(* IEC 61131-3 sources: std_i2980_v2.06_cp053/Source/IMM/ieccontrol/simulation (part 8) *)

(* ---- ABSafetySimu.pu ---- *)
IMPORT_OVER_LISTFILE
 cTimeSGAutoClose
, cTimeSGAutoOpen
, cTimeSGAutoLock
, cTimeSGAutoUnlock
, cTimeSGAutoFast
, FBEPForceDI
, FBEPUnForceDI
, ABForceDigital
, KSYS_Status
, TON

END_IMPORT

ALGORITHM_BLOCK ABSafetySimu #DUMMY_EDIT_BLOCK

SYSTEM_VAR
 sv_bInitStart : BOOL;
 sv_bSimulate : BOOL;
 sv_ForceSGMoldClose : BOOL;
 sv_ForceSGNozzleClose : BOOL;
 sv_ForceSGNozzleRearClose : BOOL;
 sv_ForceSGRearClose : BOOL;
 sv_ForceEmergencyStop1 : BOOL;
 sv_ForceEmergencyStop2 : BOOL;
 sv_ForceEmergencyStop3 : BOOL;
 sv_ForceEmergencyStop4 : BOOL;
 sv_ForceOilFilterOK : BOOL;
 sv_ForceLightCurtainClose : BOOL;
 sv_ForceSafetyMat : BOOL;
END_VAR

SYSTEM_OBJECT
 TaskSim : TASK;
 PU_Task_13 : TASK;
END_OBJECT

VAR
 fbEPForceDI : FBEPForceDI;
 fbEPUnForceDI : FBEPUnForceDI;
 mbDIEmergencyStop1Linked : BOOL;
 mbDIEmergencyStop2Linked : BOOL;
 mbDIEmergencyStop3Linked : BOOL;
 mbDIEmergencyStop4Linked : BOOL;
 mbDIOilFilterOkLinked : BOOL;
 mbDISGNozzleLinked : BOOL;
 mbDISGNozzleRearLinked : BOOL;
 mbDISGRearLinked : BOOL;
 mbDISGMoldLinked : BOOL;
 mbDISGMoldOpenLinked : BOOL;
 mpbDISGAutoClosed1 : REFTO BOOL;
 mbDISGAutoClosed1Linked : BOOL;
 mpbDISGAutoClosed2 : REFTO BOOL;
 mbDISGAutoClosed2Linked : BOOL;
 mpbDISGAutoOpen : REFTO BOOL;
 mbDISGAutoOpenLinked : BOOL;
 mpbDISGAutoCloseSlow : REFTO BOOL;
 mbDISGAutoCloseSlowLinked : BOOL;
 mbDISGAutoOpenSlowLinked : BOOL;
 mpbDISGAutoLocked : REFTO BOOL;
 mbDISGAutoLockedLinked : BOOL;
 mpbDISGAutoUnlocked : REFTO BOOL;
 mbDISGAutoUnlockedLinked : BOOL;
 mpbDOSGAutoClose : REFTO BOOL;
 mbDOSGAutoCloseLinked : BOOL;
 mpbDOSGAutoFast : REFTO BOOL;
 mbDOSGAutoFastLinked : BOOL;
 mpbDOSGAutoOpen : REFTO BOOL;
 mbDOSGAutoOpenLinked : BOOL;
 mpbDOSGAutoLock : REFTO BOOL;
 mbDOSGAutoLockLinked : BOOL;
 mpbDOSGAutoUnlock : REFTO BOOL;
 mbDOSGAutoUnlockLinked : BOOL;
 mbDISafetyMat1Linked : BOOL;
 mbDISafetyMat2Linked : BOOL;
 mbDILightCurtainClosedLinked : BOOL;
END_VAR

POSTUPDATE_ALGORITHM pStart ON PU_Task_13 WITH sv_bSimulate,sv_bInitStart

#BEGIN_EDIT_BLOCK
(**************************************** WARNING ********************************************
 *** The KEBA Kemro K2 System including software is not intended for safety control tasks! ***
 ***                       For further information see Comment tab!                        ***
 *********************************************************************************************)

IF sv_bSimulate THEN
   START_PROCESS_ALGORITHM(paSimulate);
END_IF;

IF sv_bSimulate AND mbDISGAutoClosed1Linked THEN
   START_PROCESS_ALGORITHM(paSimulateSGAuto);
END_IF;

;#END_EDIT_BLOCK END_ALGORITHM

PROCESS_ALGORITHM paSimulate ON TaskSim

VAR
 fbEPUnForceDI : FBEPUnForceDI;
 mFirstTimeRun : BOOL := TRUE;
 abForceMoldOpenMaxLimitSwitch : ABForceDigital;
 abForceMoldCloseMinLimitSwitch : ABForceDigital;
END_VAR

(* IecGraph-Code *)

(* init step *)
INITIAL_STEP INIT:
aInit (P);
END_STEP

(* steps *)
STEP SIM:
aSimulate (N);
END_STEP

STEP STOP:
aStopSimu (P);
END_STEP

(* transitions *)
TRANSITION SimRequired (* Trans11 *) FROM INIT TO SIM :=  #BEGIN_EDIT_BLOCK
sv_bSimulate
;#END_EDIT_BLOCK
END_TRANSITION

TRANSITION StpSimRequired (* Trans13 *) FROM SIM TO STOP :=  #BEGIN_EDIT_BLOCK
NOT sv_bSimulate
;#END_EDIT_BLOCK
END_TRANSITION

TRANSITION Return (* Trans16 *) FROM STOP TO SIM :=  #BEGIN_EDIT_BLOCK
TRUE
;#END_EDIT_BLOCK
END_TRANSITION

(* end IecGraph-Code *)
(* sfc-code *)

(* stand alone actions *)
ACTION aSimulate: #BEGIN_EDIT_BLOCK
(**************************************** WARNING ********************************************
 *** The KEBA Kemro K2 System including software is not intended for safety control tasks! ***
 ***                       For further information see Comment tab!                        ***
 *********************************************************************************************)

IF mFirstTimeRun THEN
   sv_ForceSGMoldClose := TRUE;
   sv_ForceSGNozzleClose := TRUE;
   sv_ForceSGNozzleRearClose := TRUE;
   sv_ForceSGRearClose := TRUE;
   sv_ForceEmergencyStop1 := TRUE;
   sv_ForceEmergencyStop2 := TRUE;
   sv_ForceEmergencyStop3 := TRUE;
   sv_ForceEmergencyStop4 := TRUE;
   sv_ForceOilFilterOK := FALSE;
   sv_ForceLightCurtainClose := TRUE;
   sv_ForceSafetyMat := TRUE;
   abForceMoldOpenMaxLimitSwitch.aSetForceValue(TRUE);
   abForceMoldCloseMinLimitSwitch.aSetForceValue(TRUE);
   mFirstTimeRun := FALSE;
END_IF;

;#END_EDIT_BLOCK END_ACTION (*aSimulate*)
ACTION aStopSimu: #BEGIN_EDIT_BLOCK
IF mbDIEmergencyStop1Linked THEN
   fbEPUnForceDI(sSysVar := 'OperationMode1.di_EmergencyStop1');
END_IF;
IF mbDIEmergencyStop2Linked THEN
   fbEPUnForceDI(sSysVar := 'OperationMode1.di_EmergencyStop2');
END_IF;
IF mbDIEmergencyStop3Linked THEN
   fbEPUnForceDI(sSysVar := 'OperationMode1.di_EmergencyStop3');
END_IF;
IF mbDIEmergencyStop4Linked THEN
   fbEPUnForceDI(sSysVar := 'OperationMode1.di_EmergencyStop4');
END_IF;

IF mbDIOilFilterOkLinked THEN
   fbEPUnForceDI(sSysVar := 'OilMaintenance1.di_OilFilterOK');
END_IF;

// SG nozzle
IF mbDISGNozzleLinked THEN
   fbEPUnForceDI(sSysVar := 'SafetyGateNozzle1.di_Closed');
END_IF;

// SG nozzle rear
IF mbDISGNozzleRearLinked THEN
   fbEPUnForceDI(sSysVar := 'SafetyGateNozzleRear1.di_Closed');
END_IF;

// SG rear
IF mbDISGRearLinked THEN
   fbEPUnForceDI(sSysVar := 'SafetyGateRear1.di_Closed');
END_IF;

// SG mold
IF mbDISGMoldLinked THEN
   fbEPUnForceDI(sSysVar := 'SafetyGateMold1.di_Closed');
END_IF;
IF mbDISGMoldOpenLinked THEN
   fbEPUnForceDI(sSysVar := 'SafetyGateMold1.di_Open');
END_IF;

IF mbDISafetyMat1Linked THEN
   fbEPUnForceDI(sSysVar := 'SafetyMat1.di_SafetyMat');
END_IF;
IF mbDISafetyMat2Linked THEN
   fbEPUnForceDI(sSysVar := 'SafetyMat2.di_SafetyMat');
END_IF;

IF mbDILightCurtainClosedLinked THEN
   fbEPUnForceDI(sSysVar := 'LightCurtain1.di_Closed');
END_IF;

abForceMoldOpenMaxLimitSwitch.aUnforce();
abForceMoldCloseMinLimitSwitch.aUnforce();

mFirstTimeRun := TRUE;
STOP_PROCESS_ALGORITHM();

;#END_EDIT_BLOCK END_ACTION (*aStopSimu*)
ACTION aInit: #BEGIN_EDIT_BLOCK
(**************************************** WARNING ********************************************
 *** The KEBA Kemro K2 System including software is not intended for safety control tasks! ***
 ***                       For further information see Comment tab!                        ***
 *********************************************************************************************)

abForceMoldOpenMaxLimitSwitch.aInit('Mold1.di_MoldOpenProtect');
abForceMoldCloseMinLimitSwitch.aInit('Mold1.di_MoldCloseProtect');

;#END_EDIT_BLOCK END_ACTION (*aInit*)
(* end sfc-code *)

END_ALGORITHM

POSTUPDATE_ALGORITHM pEmergencyStop ON TaskSim WITH sv_ForceEmergencyStop1,sv_ForceEmergencyStop2,sv_ForceEmergencyStop3,sv_ForceEmergencyStop4,sv_bSimulate

#BEGIN_EDIT_BLOCK
IF sv_bSimulate THEN
   IF mbDIEmergencyStop1Linked THEN
      fbEPForceDI(sSysVar := 'OperationMode1.di_EmergencyStop1', Value := sv_ForceEmergencyStop1);
   END_IF;
   IF mbDIEmergencyStop2Linked THEN
      fbEPForceDI(sSysVar := 'OperationMode1.di_EmergencyStop2', Value := sv_ForceEmergencyStop2);
   END_IF;
   IF mbDIEmergencyStop3Linked THEN
      fbEPForceDI(sSysVar := 'OperationMode1.di_EmergencyStop3', Value := sv_ForceEmergencyStop3);
   END_IF;
   IF mbDIEmergencyStop4Linked THEN
      fbEPForceDI(sSysVar := 'OperationMode1.di_EmergencyStop4', Value := sv_ForceEmergencyStop4);
   END_IF;
END_IF;

;#END_EDIT_BLOCK END_ALGORITHM

POSTUPDATE_ALGORITHM pOilFilterOK ON TaskSim WITH sv_ForceOilFilterOK,sv_bSimulate

#BEGIN_EDIT_BLOCK
IF mbDIOilFilterOkLinked THEN
   IF sv_bSimulate THEN
      fbEPForceDI(sSysVar := 'OilMaintenance1.di_OilFilterOK', Value := sv_ForceOilFilterOK);
   END_IF;
END_IF;

;#END_EDIT_BLOCK END_ALGORITHM

POSTUPDATE_ALGORITHM pSGMoldClose ON TaskSim WITH sv_ForceSGMoldClose,sv_bSimulate

#BEGIN_EDIT_BLOCK
IF sv_bSimulate THEN
   IF mbDISGMoldLinked THEN
      fbEPForceDI(sSysVar :='SafetyGateMold1.di_Closed', Value := sv_ForceSGMoldClose);
   END_IF;
   IF mbDISGMoldOpenLinked THEN
      fbEPForceDI(sSysVar := 'SafetyGateMold1.di_Open', Value := NOT sv_ForceSGMoldClose);
   END_IF;
END_IF;

;#END_EDIT_BLOCK END_ALGORITHM

POSTUPDATE_ALGORITHM pSGNozzleClose ON TaskSim WITH sv_ForceSGNozzleClose,sv_bSimulate

#BEGIN_EDIT_BLOCK
IF sv_bSimulate THEN
   IF mbDISGNozzleLinked THEN
      fbEPForceDI(sSysVar :='SafetyGateNozzle1.di_Closed', Value := sv_ForceSGNozzleClose);
   END_IF;
END_IF;

;#END_EDIT_BLOCK END_ALGORITHM

POSTUPDATE_ALGORITHM pSGNozzleRearClose ON TaskSim WITH sv_ForceSGNozzleRearClose,sv_bSimulate

#BEGIN_EDIT_BLOCK
IF sv_bSimulate THEN
   IF mbDISGNozzleRearLinked THEN
      fbEPForceDI(sSysVar :='SafetyGateNozzleRear1.di_Closed', Value := sv_ForceSGNozzleRearClose);
   END_IF;
END_IF;

;#END_EDIT_BLOCK END_ALGORITHM

POSTUPDATE_ALGORITHM pSGRearClose ON TaskSim WITH sv_ForceSGRearClose,sv_bSimulate

#BEGIN_EDIT_BLOCK
IF sv_bSimulate THEN
   IF mbDISGRearLinked THEN
      fbEPForceDI(sSysVar :='SafetyGateRear1.di_Closed', Value := sv_ForceSGRearClose);
   END_IF;
END_IF;

;#END_EDIT_BLOCK END_ALGORITHM

POSTUPDATE_ALGORITHM pLightCurtainClose ON TaskSim WITH sv_ForceLightCurtainClose,sv_bSimulate

#BEGIN_EDIT_BLOCK
IF sv_bSimulate THEN
   IF mbDILightCurtainClosedLinked THEN
      fbEPForceDI(sSysVar :='LightCurtain1.di_Closed', Value := sv_ForceLightCurtainClose);
   END_IF;
END_IF;

;#END_EDIT_BLOCK END_ALGORITHM

POSTUPDATE_ALGORITHM pSafetyMat ON TaskSim WITH sv_ForceSafetyMat,sv_bSimulate

#BEGIN_EDIT_BLOCK
IF sv_bSimulate THEN
   IF mbDISafetyMat1Linked THEN
      fbEPForceDI(sSysVar :='SafetyMat1.di_SafetyMat', Value := sv_ForceSafetyMat);
   END_IF;
   IF mbDISafetyMat2Linked THEN
      fbEPForceDI(sSysVar :='SafetyMat2.di_SafetyMat', Value := sv_ForceSafetyMat);
   END_IF;
END_IF;

;#END_EDIT_BLOCK END_ALGORITHM

PROCESS_ALGORITHM paInit ON TaskSim AUTOSTART

VAR
 Status : KSYS_Status;
 pbDummy : REFTO BOOL;
END_VAR
#BEGIN_EDIT_BLOCK
pbDummy := GET_SYNC_REFTO('OperationMode1.di_EmergencyStop1', T#0s, Status);
mbDIEmergencyStop1Linked := (Status = KSYS_Status_OK);
pbDummy := GET_SYNC_REFTO('OperationMode1.di_EmergencyStop2', T#0s, Status);
mbDIEmergencyStop2Linked := (Status = KSYS_Status_OK);
pbDummy := GET_SYNC_REFTO('OperationMode1.di_EmergencyStop3', T#0s, Status);
mbDIEmergencyStop3Linked := (Status = KSYS_Status_OK);
pbDummy := GET_SYNC_REFTO('OperationMode1.di_EmergencyStop4', T#0s, Status);
mbDIEmergencyStop4Linked := (Status = KSYS_Status_OK);

pbDummy := GET_SYNC_REFTO('OilMaintenance1.di_OilFilterOK', T#0s, Status);
mbDIOilFilterOkLinked := (Status = KSYS_Status_OK);

pbDummy := GET_SYNC_REFTO('SafetyGateNozzle1.di_Closed', T#0s, Status);
mbDISGNozzleLinked := (Status = KSYS_Status_OK);

(*Optional Safety Gate Nozzle Rear*)
pbDummy := GET_SYNC_REFTO('SafetyGateNozzleRear1.di_Closed', T#0s, Status);
mbDISGNozzleRearLinked := (Status = KSYS_Status_OK);

// Safety Gate Rear
pbDummy := GET_SYNC_REFTO('SafetyGateRear1.di_Closed', T#0s, Status);
mbDISGRearLinked := (Status = KSYS_Status_OK);

// Safety Gate Mold
pbDummy := GET_SYNC_REFTO('SafetyGateMold1.di_Closed', T#0s, Status);
mbDISGMoldLinked := (Status = KSYS_Status_OK);
pbDummy := GET_SYNC_REFTO('SafetyGateMold1.di_Open', T#0s, Status);
mbDISGMoldOpenLinked := (Status = KSYS_Status_OK);

// SafetyGateAuto
mpbDISGAutoClosed1 := GET_SYNC_REFTO('SafetyGateAuto1.di_Closed', T#0s, Status);
mbDISGAutoClosed1Linked := (Status = KSYS_Status_OK);

mpbDISGAutoClosed2 := GET_SYNC_REFTO('SafetyGateAuto1.di_Closed2', T#0s, Status);
mbDISGAutoClosed2Linked := (Status = KSYS_Status_OK);

mpbDISGAutoOpen := GET_SYNC_REFTO('SafetyGateAuto1.di_Open', T#0s, Status);
mbDISGAutoOpenLinked := (Status = KSYS_Status_OK);

mpbDISGAutoCloseSlow := GET_SYNC_REFTO('SafetyGateAuto1.di_CloseSlow', T#0s, Status);
mbDISGAutoCloseSlowLinked := (Status = KSYS_Status_OK);

pbDummy := GET_SYNC_REFTO('SafetyGateAuto1.di_OpenSlow', T#0s, Status);
mbDISGAutoOpenSlowLinked := (Status = KSYS_Status_OK);

mpbDISGAutoLocked := GET_SYNC_REFTO('SafetyGateAuto1.di_Locked', T#0s, Status);
mbDISGAutoLockedLinked := (Status = KSYS_Status_OK);

mpbDISGAutoUnlocked := GET_SYNC_REFTO('SafetyGateAuto1.di_Unlocked', T#0s, Status);
mbDISGAutoUnlockedLinked := (Status = KSYS_Status_OK);

mpbDOSGAutoClose := GET_SYNC_REFTO('SafetyGateAuto1.do_Close', T#0s, Status);
mbDOSGAutoCloseLinked := (Status = KSYS_Status_OK);

mpbDOSGAutoFast := GET_SYNC_REFTO('SafetyGateAuto1.do_Fast', T#0s, Status);
mbDOSGAutoFastLinked := (Status = KSYS_Status_OK);

mpbDOSGAutoOpen := GET_SYNC_REFTO('SafetyGateAuto1.do_Open', T#0s, Status);
mbDOSGAutoOpenLinked := (Status = KSYS_Status_OK);

mpbDOSGAutoLock := GET_SYNC_REFTO('SafetyGateAuto1.do_Lock', T#0s, Status);
mbDOSGAutoLockLinked := (Status = KSYS_Status_OK);

mpbDOSGAutoUnlock := GET_SYNC_REFTO('SafetyGateAuto1.do_Unlock', T#0s, Status);
mbDOSGAutoUnlockLinked := (Status = KSYS_Status_OK);

// SafetyMat
pbDummy := GET_SYNC_REFTO('SafetyMat1.di_SafetyMat', T#0s, Status);
mbDISafetyMat1Linked := (Status = KSYS_Status_OK);

pbDummy := GET_SYNC_REFTO('SafetyMat2.di_SafetyMat', T#0s, Status);
mbDISafetyMat2Linked := (Status = KSYS_Status_OK);

//LightCurtain
pbDummy:= GET_SYNC_REFTO('LightCurtain1.di_Closed', T#0s, Status);
mbDILightCurtainClosedLinked := (Status = KSYS_Status_OK);

STOP_PROCESS_ALGORITHM();

;#END_EDIT_BLOCK END_ALGORITHM

PROCESS_ALGORITHM paSimulateSGAuto ON TaskSim

VAR
 fbTimerSGAutoClose : TON;
 fbTimerSGAutoOpen : TON;
 fbTimerSGAutoLock : TON;
 fbTimerSGAutoUnlock : TON;
 fbTimerSGAutoFast : TON;
 bInitDone : BOOL;
END_VAR

(* IecGraph-Code *)

(* init step *)
INITIAL_STEP INIT:
END_STEP

(* steps *)
STEP SIM:
aSimulate (N);
END_STEP

STEP STOP:
aStopSimu (P);
END_STEP

(* transitions *)
TRANSITION SimRequired (* Trans11 *) FROM INIT TO SIM :=  #BEGIN_EDIT_BLOCK
sv_bSimulate
;#END_EDIT_BLOCK
END_TRANSITION

TRANSITION StpSimRequired (* Trans13 *) FROM SIM TO STOP :=  #BEGIN_EDIT_BLOCK
NOT sv_bSimulate
;#END_EDIT_BLOCK
END_TRANSITION

TRANSITION Return (* Trans16 *) FROM STOP TO SIM :=  #BEGIN_EDIT_BLOCK
TRUE
;#END_EDIT_BLOCK
END_TRANSITION

(* end IecGraph-Code *)
(* sfc-code *)

(* stand alone actions *)
ACTION aStopSimu: #BEGIN_EDIT_BLOCK
IF mbDISGAutoClosed1Linked THEN
   fbEPUnForceDI(sSysVar := 'SafetyGateAuto1.di_Closed');
END_IF;

IF mbDISGAutoClosed2Linked THEN
   fbEPUnForceDI(sSysVar := 'SafetyGateAuto1.di_Closed2');
END_IF;

IF mbDISGAutoOpenLinked THEN
   fbEPUnForceDI(sSysVar := 'SafetyGateAuto1.di_Open');
END_IF;

IF mbDISGAutoOpenSlowLinked THEN
   fbEPUnForceDI(sSysVar := 'SafetyGateAuto1.di_OpenSlow');
END_IF;

IF mbDISGAutoCloseSlowLinked THEN
   fbEPUnForceDI(sSysVar := 'SafetyGateAuto1.di_CloseSlow');
END_IF;

IF mbDISGAutoLockedLinked THEN
   fbEPUnForceDI(sSysVar := 'SafetyGateAuto1.di_Locked');
END_IF;

IF mbDISGAutoUnlockedLinked THEN
   fbEPUnForceDI(sSysVar := 'SafetyGateAuto1.di_Unlocked');
END_IF;

STOP_PROCESS_ALGORITHM();

;#END_EDIT_BLOCK END_ACTION (*aStopSimu*)
ACTION aSimulate: #BEGIN_EDIT_BLOCK
//-------------------------------------------//
// normal movement simulation                //
//-------------------------------------------//

IF NOT bInitDone THEN
   fbEPForceDI(sSysVar := 'SafetyGateAuto1.di_Emergency',Value := TRUE);
   fbEPForceDI(sSysVar := 'SafetyGateAuto1.di_Emergency2',Value := TRUE);

   IF mbDISGAutoClosed1Linked THEN
      fbEPForceDI(sSysVar :='SafetyGateAuto1.di_Closed', Value := FALSE);
   END_IF;
   IF mbDISGAutoClosed2Linked THEN
      fbEPForceDI(sSysVar :='SafetyGateAuto1.di_Closed2', Value := TRUE);
   END_IF;
   IF mbDISGAutoCloseSlowLinked THEN
      fbEPForceDI(sSysVar :='SafetyGateAuto1.di_CloseSlow', Value := FALSE);
   END_IF;

   IF mbDISGAutoOpenLinked THEN
      fbEPForceDI(sSysVar :='SafetyGateAuto1.di_Open', Value := TRUE);
   END_IF;
   IF mbDISGAutoOpenSlowLinked THEN
      fbEPForceDI(sSysVar :='SafetyGateAuto1.di_OpenSlow', Value := TRUE);
   END_IF;

   IF mbDISGAutoLockedLinked THEN
      fbEPForceDI(sSysVar :='SafetyGateAuto1.di_Locked', Value := TRUE);
   END_IF;
   IF mbDISGAutoUnlockedLinked THEN
      fbEPForceDI(sSysVar :='SafetyGateAuto1.di_Unlocked', Value := FALSE);
   END_IF;

   bInitDone := TRUE;
END_IF;

// Safety Gate Close
IF mbDOSGAutoCloseLinked AND mpbDOSGAutoClose^ THEN

   IF mbDISGAutoOpenLinked AND mpbDISGAutoOpen^ THEN
      fbEPForceDI(sSysVar := 'SafetyGateAuto1.di_Open',Value := FALSE);
      fbEPForceDI(sSysVar := 'SafetyGateAuto1.di_OpenSlow',Value := FALSE);
   END_IF;

   IF mbDOSGAutoFastLinked THEN
       fbTimerSGAutoFast (IN := mpbDOSGAutoFast^,
                      PT := cTimeSGAutoFast);
   END_IF;
   IF fbTimerSGAutoFast.Q THEN
      fbTimerSGAutoFast(IN := FALSE);
      fbEPForceDI(sSysVar := 'SafetyGateAuto1.di_CloseSlow',Value := TRUE);
   END_IF;

   fbTimerSGAutoClose (IN := mpbDOSGAutoClose^,
                       PT := cTimeSGAutoClose);
   IF fbTimerSGAutoClose.Q THEN
      fbTimerSGAutoClose(IN := FALSE);
      fbEPForceDI(sSysVar := 'SafetyGateAuto1.di_Closed',Value := TRUE);
      fbEPForceDI(sSysVar := 'SafetyGateAuto1.di_Closed2',Value := FALSE);
   END_IF;
END_IF;

// Safety Gate Open
IF mbDOSGAutoOpenLinked AND mpbDOSGAutoOpen^ THEN
   IF mbDISGAutoClosed1Linked AND mpbDISGAutoClosed1^ THEN
      fbEPForceDI(sSysVar := 'SafetyGateAuto1.di_Closed',Value := FALSE);
      fbEPForceDI(sSysVar := 'SafetyGateAuto1.di_CloseSlow',Value := FALSE);
   END_IF;

   IF mbDISGAutoClosed2Linked AND NOT mpbDISGAutoClosed2^ THEN
      fbEPForceDI(sSysVar := 'SafetyGateAuto1.di_Closed2',Value := TRUE);
   END_IF;

   IF mbDOSGAutoFastLinked THEN
   fbTimerSGAutoFast (IN := mpbDOSGAutoFast^,
                      PT := cTimeSGAutoFast);
   END_IF;
   IF fbTimerSGAutoFast.Q THEN
      fbTimerSGAutoFast(IN := FALSE);
      fbEPForceDI(sSysVar := 'SafetyGateAuto1.di_OpenSlow',Value := TRUE);
   END_IF;

   fbTimerSGAutoOpen (IN := mpbDOSGAutoOpen^,
                       PT := cTimeSGAutoOpen);
   IF fbTimerSGAutoOpen.Q THEN
      fbTimerSGAutoOpen(IN := FALSE);
      fbEPForceDI(sSysVar := 'SafetyGateAuto1.di_Open',Value := TRUE);
   END_IF;
END_IF;

// Safety Gate Lock
IF mbDOSGAutoLockLinked AND mpbDOSGAutoLock^ THEN
   IF mbDISGAutoUnlockedLinked AND mpbDISGAutoUnlocked^ THEN
      fbEPForceDI(sSysVar := 'SafetyGateAuto1.di_Unlocked',Value := FALSE);
   END_IF;

   fbTimerSGAutoLock (IN := mpbDOSGAutoLock^,
                      PT := cTimeSGAutoLock);
   IF fbTimerSGAutoLock.Q THEN
      fbTimerSGAutoLock(IN := TRUE);
      fbEPForceDI(sSysVar := 'SafetyGateAuto1.di_Locked',Value := TRUE);
   END_IF;
END_IF;

// Safety Gate Unlock
IF mbDOSGAutoUnlockLinked AND mpbDOSGAutoUnlock^ THEN
   IF mbDISGAutoLockedLinked AND mpbDISGAutoLocked^ THEN
      fbEPForceDI(sSysVar := 'SafetyGateAuto1.di_Locked',Value := FALSE);
   END_IF;

   fbTimerSGAutoUnlock (IN := mpbDOSGAutoUnlock^,
                        PT := cTimeSGAutoUnlock);
   IF fbTimerSGAutoUnlock.Q THEN
      fbTimerSGAutoUnlock(IN := TRUE);
      fbEPForceDI(sSysVar := 'SafetyGateAuto1.di_Unlocked',Value := TRUE);
   END_IF;
END_IF;

;#END_EDIT_BLOCK END_ACTION (*aSimulate*)
(* end sfc-code *)

END_ALGORITHM

END_ALGORITHM_BLOCK

#END_OF_IEC_PART

@Puma @IecEditor 6 97 @Pou 25
@@@BEG_Comment@@@

@@@END_Comment@@@

@BEG_Contents

@BEG_Func
@RT(17)FuncTreeContainer
0
@END_Func

@BEG_Const
@RT(18)ConstTreeContainer
5
@Var @RT(16)cTimeSGAutoClose @RT(0) @T @F @DT @RT(4)TIME @RT(0) @T @T @BASIC 0 @F
@F @F
@T
@BEG_Attrib
0 @RT(4)t#3s @RT(0)
@END_Attrib
1 1 @F @F @F @F

@Var @RT(15)cTimeSGAutoOpen @RT(0) @T @F @DT @RT(4)TIME @RT(0) @T @T @BASIC 0 @F
@F @F
@T
@BEG_Attrib
0 @RT(4)t#3s @RT(0)
@END_Attrib
1 1 @F @F @F @F

@Var @RT(15)cTimeSGAutoLock @RT(0) @T @F @DT @RT(4)TIME @RT(0) @T @T @BASIC 0 @F
@F @F
@T
@BEG_Attrib
0 @RT(4)t#1s @RT(0)
@END_Attrib
1 1 @F @F @F @F

@Var @RT(17)cTimeSGAutoUnlock @RT(0) @T @F @DT @RT(4)TIME @RT(0) @T @T @BASIC 0 @F
@F @F
@T
@BEG_Attrib
0 @RT(4)t#1s @RT(0)
@END_Attrib
1 1 @F @F @F @F

@Var @RT(15)cTimeSGAutoFast @RT(0) @T @F @DT @RT(4)TIME @RT(0) @T @T @BASIC 0 @F
@F @F
@T
@BEG_Attrib
0 @RT(4)t#2s @RT(0)
@END_Attrib
1 1 @F @F @F @F

@END_Const

@BEG_Export

@BEG_Kind
@ALGORITHM_BLOCK @RT(12)ABSafetySimu @STRUCTURED_TEXT
@RT(0) @RT(0) @RT(0)
@END_Kind

@BEG_Dcl
@RT(16)DclTreeContainer
53
@Var @RT(7)TaskSim @RT(0) @T @T @RENAMED 0 @T @T @DT @RT(4)TASK @RT(0) @T @T @BASIC 0 @F
@F @F
@T
@BEG_Attrib
3 @RT(0) @RT(0) @RT(0)
@END_Attrib
1 7 @F @F @F @F

@Var @RT(10)PU_Task_13 @RT(0) @T @T @RENAMED 0 @T @T @DT @RT(4)TASK @RT(0) @T @T @BASIC 0 @F
@F @F
@T
@BEG_Attrib
3 @RT(0) @RT(0) @RT(0)
@END_Attrib
1 7 @F @F @F @F

@Var @RT(13)sv_bInitStart @RT(0) @T @F @DT @RT(4)BOOL @RT(0) @T @T @BASIC 0 @F
@F @F
@T
@BEG_Attrib
3 @RT(0) @RT(0) @RT(0)
@END_Attrib
1 8 @F @F @F @F

@Var @RT(12)sv_bSimulate @RT(0) @T @F @DT @RT(4)BOOL @RT(0) @T @T @BASIC 0 @F
@F @F
@T
@BEG_Attrib
3 @RT(0) @RT(0) @RT(0)
@END_Attrib
1 8 @F @F @F @F

@Var @RT(11)fbEPForceDI @RT(0) @T @T @DERIVED 0 @T @T @DT @RT(11)FBEPForceDI @RT(0) @T @T @UNKNOWN 0 @F
@F @F
@T
@BEG_Attrib
3 @RT(0) @RT(0) @RT(0)
@END_Attrib
1 0 @F @F @F @F

@Var @RT(13)fbEPUnForceDI @RT(0) @T @T @DERIVED 0 @T @T @DT @RT(13)FBEPUnForceDI @RT(0) @T @T @UNKNOWN 0 @F
@F @F
@T
@BEG_Attrib
3 @RT(0) @RT(0) @RT(0)
@END_Attrib
1 0 @F @F @F @F

@Var @RT(19)sv_ForceSGMoldClose @RT(0) @T @F @DT @RT(4)BOOL @RT(0) @T @T @BASIC 0 @F
@F @F
@T
@BEG_Attrib
3 @RT(0) @RT(0) @RT(0)
@END_Attrib
1 8 @F @F @F @F

@Var @RT(21)sv_ForceSGNozzleClose @RT(0) @T @F @DT @RT(4)BOOL @RT(0) @T @T @BASIC 0 @F
@F @F
@T
@BEG_Attrib
3 @RT(0) @RT(0) @RT(0)
@END_Attrib
1 8 @F @F @F @F

@Var @RT(25)sv_ForceSGNozzleRearClose @RT(0) @T @F @DT @RT(4)BOOL @RT(0) @T @T @BASIC 0 @F
@F @F
@T
@BEG_Attrib
3 @RT(0) @RT(0) @RT(0)
@END_Attrib
1 8 @F @F @F @F

@Var @RT(19)sv_ForceSGRearClose @RT(0) @T @F @DT @RT(4)BOOL @RT(0) @T @T @BASIC 0 @F
@F @F
@T
@BEG_Attrib
3 @RT(0) @RT(0) @RT(0)
@END_Attrib
1 8 @F @F @F @F

@Var @RT(22)sv_ForceEmergencyStop1 @RT(0) @T @F @DT @RT(4)BOOL @RT(0) @T @T @BASIC 0 @F
@F @F
@T
@BEG_Attrib
3 @RT(0) @RT(0) @RT(0)
@END_Attrib
1 8 @F @F @F @F

@Var @RT(22)sv_ForceEmergencyStop2 @RT(0) @T @F @DT @RT(4)BOOL @RT(0) @T @T @BASIC 0 @F
@F @F
@T
@BEG_Attrib
3 @RT(0) @RT(0) @RT(0)
@END_Attrib
1 8 @F @F @F @F

@Var @RT(22)sv_ForceEmergencyStop3 @RT(0) @T @F @DT @RT(4)BOOL @RT(0) @T @T @BASIC 0 @F
@F @F
@T
@BEG_Attrib
3 @RT(0) @RT(0) @RT(0)
@END_Attrib
1 8 @F @F @F @F

@Var @RT(22)sv_ForceEmergencyStop4 @RT(0) @T @F @DT @RT(4)BOOL @RT(0) @T @T @BASIC 0 @F
@F @F
@T
@BEG_Attrib
3 @RT(0) @RT(0) @RT(0)
@END_Attrib
1 8 @F @F @F @F

@Var @RT(19)sv_ForceOilFilterOK @RT(0) @T @F @DT @RT(4)BOOL @RT(0) @T @T @BASIC 0 @F
@F @F
@T
@BEG_Attrib
3 @RT(0) @RT(0) @RT(0)
@END_Attrib
1 8 @F @F @F @F

@Var @RT(25)sv_ForceLightCurtainClose @RT(0) @T @T @RENAMED 0 @T @T @DT @RT(4)BOOL @RT(0) @T @T @BASIC 0 @F
@F @F
@T
@BEG_Attrib
3 @RT(0) @RT(0) @RT(0)
@END_Attrib
1 8 @F @F @F @F

@Var @RT(17)sv_ForceSafetyMat @RT(0) @T @T @RENAMED 0 @T @T @DT @RT(4)BOOL @RT(0) @T @T @BASIC 0 @F
@F @F
@T
@BEG_Attrib
3 @RT(0) @RT(0) @RT(0)
@END_Attrib
1 8 @F @F @F @F

@Var @RT(24)mbDIEmergencyStop1Linked @RT(0) @T @F @DT @RT(4)BOOL @RT(0) @T @T @BASIC 0 @F
@F @F
@T
@BEG_Attrib
3 @RT(0) @RT(0) @RT(0)
@END_Attrib
1 0 @F @F @F @F

@Var @RT(24)mbDIEmergencyStop2Linked @RT(0) @T @F @DT @RT(4)BOOL @RT(0) @T @T @BASIC 0 @F
@F @F
@T
@BEG_Attrib
3 @RT(0) @RT(0) @RT(0)
@END_Attrib
1 0 @F @F @F @F

@Var @RT(24)mbDIEmergencyStop3Linked @RT(0) @T @F @DT @RT(4)BOOL @RT(0) @T @T @BASIC 0 @F
@F @F
@T
@BEG_Attrib
3 @RT(0) @RT(0) @RT(0)
@END_Attrib
1 0 @F @F @F @F

@Var @RT(24)mbDIEmergencyStop4Linked @RT(0) @T @F @DT @RT(4)BOOL @RT(0) @T @T @BASIC 0 @F
@F @F
@T
@BEG_Attrib
3 @RT(0) @RT(0) @RT(0)
@END_Attrib
1 0 @F @F @F @F

@Var @RT(21)mbDIOilFilterOkLinked @RT(0) @T @F @DT @RT(4)BOOL @RT(0) @T @T @BASIC 0 @F
@F @F
@T
@BEG_Attrib
3 @RT(0) @RT(0) @RT(0)
@END_Attrib
1 0 @F @F @F @F

@Var @RT(18)mbDISGNozzleLinked @RT(0) @T @F @DT @RT(4)BOOL @RT(0) @T @T @BASIC 0 @F
@F @F
@T
@BEG_Attrib
3 @RT(0) @RT(0) @RT(0)
@END_Attrib
1 0 @F @F @F @F

@Var @RT(22)mbDISGNozzleRearLinked @RT(0) @T @F @DT @RT(4)BOOL @RT(0) @T @T @BASIC 0 @F
@F @F
@T
@BEG_Attrib
3 @RT(0) @RT(0) @RT(0)
@END_Attrib
1 0 @F @F @F @F

@Var @RT(16)mbDISGRearLinked @RT(0) @T @F @DT @RT(4)BOOL @RT(0) @T @T @BASIC 0 @F
@F @F
@T
@BEG_Attrib
3 @RT(0) @RT(0) @RT(0)
@END_Attrib
1 0 @F @F @F @F

@Var @RT(16)mbDISGMoldLinked @RT(0) @T @F @DT @RT(4)BOOL @RT(0) @T @T @BASIC 0 @F
@F @F
@T
@BEG_Attrib
3 @RT(0) @RT(0) @RT(0)
@END_Attrib
1 0 @F @F @F @F

@Var @RT(20)mbDISGMoldOpenLinked @RT(0) @T @F @DT @RT(4)BOOL @RT(0) @T @T @BASIC 0 @F
@F @F
@T
@BEG_Attrib
3 @RT(0) @RT(0) @RT(0)
@END_Attrib
1 0 @F @F @F @F

@Var @RT(18)mpbDISGAutoClosed1 @RT(0) @T @T @REFTO 0 @T @DT @RT(4)BOOL @RT(0) @T @T @BASIC 0 @F
@F @F
@T
@BEG_Attrib
3 @RT(0) @RT(0) @RT(0)
@END_Attrib
1 0 @F @F @F @F

@Var @RT(23)mbDISGAutoClosed1Linked @RT(0) @T @F @DT @RT(4)BOOL @RT(0) @T @T @BASIC 0 @F
@F @F
@T
@BEG_Attrib
3 @RT(0) @RT(0) @RT(0)
@END_Attrib
1 0 @F @F @F @F

@Var @RT(18)mpbDISGAutoClosed2 @RT(0) @T @T @REFTO 0 @T @DT @RT(4)BOOL @RT(0) @T @T @BASIC 0 @F
@F @F
@T
@BEG_Attrib
3 @RT(0) @RT(0) @RT(0)
@END_Attrib
1 0 @F @F @F @F

@Var @RT(23)mbDISGAutoClosed2Linked @RT(0) @T @F @DT @RT(4)BOOL @RT(0) @T @T @BASIC 0 @F
@F @F
@T
@BEG_Attrib
3 @RT(0) @RT(0) @RT(0)
@END_Attrib
1 0 @F @F @F @F

@Var @RT(15)mpbDISGAutoOpen @RT(0) @T @T @REFTO 0 @T @DT @RT(4)BOOL @RT(0) @T @T @BASIC 0 @F
@F @F
@T
@BEG_Attrib
3 @RT(0) @RT(0) @RT(0)
@END_Attrib
1 0 @F @F @F @F

@Var @RT(20)mbDISGAutoOpenLinked @RT(0) @T @F @DT @RT(4)BOOL @RT(0) @T @T @BASIC 0 @F
@F @F
@T
@BEG_Attrib
3 @RT(0) @RT(0) @RT(0)
@END_Attrib
1 0 @F @F @F @F

@Var @RT(20)mpbDISGAutoCloseSlow @RT(0) @T @T @REFTO 0 @T @DT @RT(4)BOOL @RT(0) @T @T @BASIC 0 @F
@F @F
@T
@BEG_Attrib
3 @RT(0) @RT(0) @RT(0)
@END_Attrib
1 0 @F @F @F @F

@Var @RT(25)mbDISGAutoCloseSlowLinked @RT(0) @T @F @DT @RT(4)BOOL @RT(0) @T @T @BASIC 0 @F
@F @F
@T
@BEG_Attrib
3 @RT(0) @RT(0) @RT(0)
@END_Attrib
1 0 @F @F @F @F

@Var @RT(24)mbDISGAutoOpenSlowLinked @RT(0) @T @F @DT @RT(4)BOOL @RT(0) @T @T @BASIC 0 @F
@F @F
@T
@BEG_Attrib
3 @RT(0) @RT(0) @RT(0)
@END_Attrib
1 0 @F @F @F @F

@Var @RT(17)mpbDISGAutoLocked @RT(0) @T @T @REFTO 0 @T @DT @RT(4)BOOL @RT(0) @T @T @BASIC 0 @F
@F @F
@T
@BEG_Attrib
3 @RT(0) @RT(0) @RT(0)
@END_Attrib
1 0 @F @F @F @F

@Var @RT(22)mbDISGAutoLockedLinked @RT(0) @T @F @DT @RT(4)BOOL @RT(0) @T @T @BASIC 0 @F
@F @F
@T
@BEG_Attrib
3 @RT(0) @RT(0) @RT(0)
@END_Attrib
1 0 @F @F @F @F

@Var @RT(19)mpbDISGAutoUnlocked @RT(0) @T @T @REFTO 0 @T @DT @RT(4)BOOL @RT(0) @T @T @BASIC 0 @F
@F @F
@T
@BEG_Attrib
3 @RT(0) @RT(0) @RT(0)
@END_Attrib
1 0 @F @F @F @F

@Var @RT(24)mbDISGAutoUnlockedLinked @RT(0) @T @F @DT @RT(4)BOOL @RT(0) @T @T @BASIC 0 @F
@F @F
@T
@BEG_Attrib
3 @RT(0) @RT(0) @RT(0)
@END_Attrib
1 0 @F @F @F @F

@Var @RT(16)mpbDOSGAutoClose @RT(0) @T @T @REFTO 0 @T @DT @RT(4)BOOL @RT(0) @T @T @BASIC 0 @F
@F @F
@T
@BEG_Attrib
3 @RT(0) @RT(0) @RT(0)
@END_Attrib
1 0 @F @F @F @F

@Var @RT(21)mbDOSGAutoCloseLinked @RT(0) @T @F @DT @RT(4)BOOL @RT(0) @T @T @BASIC 0 @F
@F @F
@T
@BEG_Attrib
3 @RT(0) @RT(0) @RT(0)
@END_Attrib
1 0 @F @F @F @F

@Var @RT(15)mpbDOSGAutoFast @RT(0) @T @T @REFTO 0 @T @DT @RT(4)BOOL @RT(0) @T @T @BASIC 0 @F
@F @F
@T
@BEG_Attrib
3 @RT(0) @RT(0) @RT(0)
@END_Attrib
1 0 @F @F @F @F

@Var @RT(20)mbDOSGAutoFastLinked @RT(0) @T @F @DT @RT(4)BOOL @RT(0) @T @T @BASIC 0 @F
@F @F
@T
@BEG_Attrib
3 @RT(0) @RT(0) @RT(0)
@END_Attrib
1 0 @F @F @F @F

@Var @RT(15)mpbDOSGAutoOpen @RT(0) @T @T @REFTO 0 @T @DT @RT(4)BOOL @RT(0) @T @T @BASIC 0 @F
@F @F
@T
@BEG_Attrib
3 @RT(0) @RT(0) @RT(0)
@END_Attrib
1 0 @F @F @F @F

@Var @RT(20)mbDOSGAutoOpenLinked @RT(0) @T @F @DT @RT(4)BOOL @RT(0) @T @T @BASIC 0 @F
@F @F
@T
@BEG_Attrib
3 @RT(0) @RT(0) @RT(0)
@END_Attrib
1 0 @F @F @F @F

@Var @RT(15)mpbDOSGAutoLock @RT(0) @T @T @REFTO 0 @T @DT @RT(4)BOOL @RT(0) @T @T @BASIC 0 @F
@F @F
@T
@BEG_Attrib
3 @RT(0) @RT(0) @RT(0)
@END_Attrib
1 0 @F @F @F @F

@Var @RT(20)mbDOSGAutoLockLinked @RT(0) @T @F @DT @RT(4)BOOL @RT(0) @T @T @BASIC 0 @F
@F @F
@T
@BEG_Attrib
3 @RT(0) @RT(0) @RT(0)
@END_Attrib
1 0 @F @F @F @F

@Var @RT(17)mpbDOSGAutoUnlock @RT(0) @T @T @REFTO 0 @T @DT @RT(4)BOOL @RT(0) @T @T @BASIC 0 @F
@F @F
@T
@BEG_Attrib
3 @RT(0) @RT(0) @RT(0)
@END_Attrib
1 0 @F @F @F @F

@Var @RT(22)mbDOSGAutoUnlockLinked @RT(0) @T @F @DT @RT(4)BOOL @RT(0) @T @T @BASIC 0 @F
@F @F
@T
@BEG_Attrib
3 @RT(0) @RT(0) @RT(0)
@END_Attrib
1 0 @F @F @F @F

@Var @RT(20)mbDISafetyMat1Linked @RT(0) @T @F @DT @RT(4)BOOL @RT(0) @T @T @BASIC 0 @F
@F @F
@T
@BEG_Attrib
3 @RT(0) @RT(0) @RT(0)
@END_Attrib
1 0 @F @F @F @F

@Var @RT(20)mbDISafetyMat2Linked @RT(0) @T @F @DT @RT(4)BOOL @RT(0) @T @T @BASIC 0 @F
@F @F
@T
@BEG_Attrib
3 @RT(0) @RT(0) @RT(0)
@END_Attrib
1 0 @F @F @F @F

@Var @RT(28)mbDILightCurtainClosedLinked @RT(0) @T @F @DT @RT(4)BOOL @RT(0) @T @T @BASIC 0 @F
@F @F
@T
@BEG_Attrib
3 @RT(0) @RT(0) @RT(0)
@END_Attrib
1 0 @F @F @F @F

@END_Dcl

@END_Export

@BEG_Body

12

@BEG_Export

@BEG_Algo
@POSTUPDATE_ALGORITHM @RT(6)pStart @STRUCTURED_TEXT
@RT(0) @RT(26)sv_bSimulate,sv_bInitStart @RT(10)PU_Task_13 @F @F
@END_Algo

@BEG_Dcl
@RT(16)DclTreeContainer
0
@END_Dcl

@END_Export

@BEG_Export

@BEG_Algo
@PROCESS_ALGORITHM @RT(10)paSimulate @SEQUENTIAL_FLOW_CHART
@RT(0) @RT(0) @RT(7)TaskSim @F @F
@END_Algo

@BEG_Dcl
@RT(16)DclTreeContainer
4
@Var @RT(13)fbEPUnForceDI @RT(0) @T @T @DERIVED 0 @T @T @DT @RT(13)FBEPUnForceDI @RT(0) @T @T @UNKNOWN 0 @F
@F @F
@T
@BEG_Attrib
3 @RT(0) @RT(0) @RT(0)
@END_Attrib
1 0 @F @F @F @F

@Var @RT(13)mFirstTimeRun @RT(0) @T @F @DT @RT(4)BOOL @RT(0) @T @T @BASIC 0 @F
@F @F
@T
@BEG_Attrib
3 @RT(4)TRUE @RT(0) @RT(0)
@END_Attrib
1 0 @F @F @F @F

@Var @RT(29)abForceMoldOpenMaxLimitSwitch @RT(0) @T @T @DERIVED 0 @F @RT(14)ABForceDigital @F
@T
@BEG_Attrib
3 @RT(0) @RT(0) @RT(0)
@END_Attrib
1 0 @F @F @F @F

@Var @RT(30)abForceMoldCloseMinLimitSwitch @RT(0) @T @T @DERIVED 0 @F @RT(14)ABForceDigital @F
@T
@BEG_Attrib
3 @RT(0) @RT(0) @RT(0)
@END_Attrib
1 0 @F @F @F @F

@END_Dcl

@END_Export

@BEG_Export

@BEG_Algo
@POSTUPDATE_ALGORITHM @RT(14)pEmergencyStop @STRUCTURED_TEXT
@RT(0) @RT(104)sv_ForceEmergencyStop1,sv_ForceEmergencyStop2,sv_ForceEmergencyStop3,sv_ForceEmergencyStop4,sv_bSimulate @RT(7)TaskSim @F @F
@END_Algo

@BEG_Dcl
@RT(16)DclTreeContainer
0
@END_Dcl

@END_Export

@BEG_Export

@BEG_Algo
@POSTUPDATE_ALGORITHM @RT(12)pOilFilterOK @STRUCTURED_TEXT
@RT(0) @RT(32)sv_ForceOilFilterOK,sv_bSimulate @RT(7)TaskSim @F @F
@END_Algo

@BEG_Dcl
@RT(16)DclTreeContainer
0
@END_Dcl

@END_Export

@BEG_Export

@BEG_Algo
@POSTUPDATE_ALGORITHM @RT(12)pSGMoldClose @STRUCTURED_TEXT
@RT(0) @RT(32)sv_ForceSGMoldClose,sv_bSimulate @RT(7)TaskSim @F @F
@END_Algo

@BEG_Dcl
@RT(16)DclTreeContainer
0
@END_Dcl

@END_Export

@BEG_Export

@BEG_Algo
@POSTUPDATE_ALGORITHM @RT(14)pSGNozzleClose @STRUCTURED_TEXT
@RT(0) @RT(34)sv_ForceSGNozzleClose,sv_bSimulate @RT(7)TaskSim @F @F
@END_Algo

@BEG_Dcl
@RT(16)DclTreeContainer
0
@END_Dcl

@END_Export

@BEG_Export

@BEG_Algo
@POSTUPDATE_ALGORITHM @RT(18)pSGNozzleRearClose @STRUCTURED_TEXT
@RT(0) @RT(38)sv_ForceSGNozzleRearClose,sv_bSimulate @RT(7)TaskSim @F @F
@END_Algo

@BEG_Dcl
@RT(16)DclTreeContainer
0
@END_Dcl

@END_Export

@BEG_Export

@BEG_Algo
@POSTUPDATE_ALGORITHM @RT(12)pSGRearClose @STRUCTURED_TEXT
@RT(0) @RT(32)sv_ForceSGRearClose,sv_bSimulate @RT(7)TaskSim @F @F
@END_Algo

@BEG_Dcl
@RT(16)DclTreeContainer
0
@END_Dcl

@END_Export

@BEG_Export

@BEG_Algo
@POSTUPDATE_ALGORITHM @RT(18)pLightCurtainClose @STRUCTURED_TEXT
@RT(0) @RT(38)sv_ForceLightCurtainClose,sv_bSimulate @RT(7)TaskSim @F @F
@END_Algo

@BEG_Dcl
@RT(16)DclTreeContainer
0
@END_Dcl

@END_Export

@BEG_Export

@BEG_Algo
@POSTUPDATE_ALGORITHM @RT(10)pSafetyMat @STRUCTURED_TEXT
@RT(0) @RT(30)sv_ForceSafetyMat,sv_bSimulate @RT(7)TaskSim @F @F
@END_Algo

@BEG_Dcl
@RT(16)DclTreeContainer
0
@END_Dcl

@END_Export

@BEG_Export

@BEG_Algo
@PROCESS_ALGORITHM @RT(6)paInit @STRUCTURED_TEXT
@RT(0) @RT(0) @RT(7)TaskSim @T @F
@END_Algo

@BEG_Dcl
@RT(16)DclTreeContainer
2
@Var @RT(6)Status @RT(0) @T @T @DERIVED 0 @T @T @DT @RT(11)KSYS_Status @RT(0) @T @T @UNKNOWN 0 @F
@F @F
@T
@BEG_Attrib
3 @RT(0) @RT(0) @RT(0)
@END_Attrib
1 0 @F @F @F @F

@Var @RT(7)pbDummy @RT(0) @T @T @REFTO 0 @T @DT @RT(4)BOOL @RT(0) @T @T @BASIC 0 @F
@F @F
@T
@BEG_Attrib
3 @RT(0) @RT(0) @RT(0)
@END_Attrib
1 0 @F @F @F @F

@END_Dcl

@END_Export

@BEG_Export

@BEG_Algo
@PROCESS_ALGORITHM @RT(16)paSimulateSGAuto @SEQUENTIAL_FLOW_CHART
@RT(0) @RT(0) @RT(7)TaskSim @F @F
@END_Algo

@BEG_Dcl
@RT(16)DclTreeContainer
6
@Var @RT(18)fbTimerSGAutoClose @RT(0) @T @T @DERIVED 0 @T @T @DT @RT(3)TON @RT(0) @T @T @UNKNOWN 0 @F
@F @F
@T
@BEG_Attrib
3 @RT(0) @RT(0) @RT(0)
@END_Attrib
1 0 @F @F @F @F

@Var @RT(17)fbTimerSGAutoOpen @RT(0) @T @T @DERIVED 0 @T @T @DT @RT(3)TON @RT(0) @T @T @UNKNOWN 0 @F
@F @F
@T
@BEG_Attrib
3 @RT(0) @RT(0) @RT(0)
@END_Attrib
1 0 @F @F @F @F

@Var @RT(17)fbTimerSGAutoLock @RT(0) @T @T @DERIVED 0 @T @T @DT @RT(3)TON @RT(0) @T @T @UNKNOWN 0 @F
@F @F
@T
@BEG_Attrib
3 @RT(0) @RT(0) @RT(0)
@END_Attrib
1 0 @F @F @F @F

@Var @RT(19)fbTimerSGAutoUnlock @RT(0) @T @T @DERIVED 0 @T @T @DT @RT(3)TON @RT(0) @T @T @UNKNOWN 0 @F
@F @F
@T
@BEG_Attrib
3 @RT(0) @RT(0) @RT(0)
@END_Attrib
1 0 @F @F @F @F

@Var @RT(17)fbTimerSGAutoFast @RT(0) @T @T @DERIVED 0 @T @T @DT @RT(3)TON @RT(0) @T @T @UNKNOWN 0 @F
@F @F
@T
@BEG_Attrib
3 @RT(0) @RT(0) @RT(0)
@END_Attrib
1 0 @F @F @F @F

@Var @RT(9)bInitDone @RT(0) @T @F @DT @RT(4)BOOL @RT(0) @T @T @BASIC 0 @F
@F @F
@T
@BEG_Attrib
3 @RT(0) @RT(0) @RT(0)
@END_Attrib
1 0 @F @F @F @F

@END_Dcl

@END_Export

@BEG_Body
@TL(13)
(**************************************** WARNING ********************************************
 *** The KEBA Kemro K2 System including software is not intended for safety control tasks! ***
 ***                       For further information see Comment tab!                        ***
 *********************************************************************************************)

IF sv_bSimulate THEN
   START_PROCESS_ALGORITHM(paSimulate);
END_IF;

IF sv_bSimulate AND mbDISGAutoClosed1Linked THEN
   START_PROCESS_ALGORITHM(paSimulateSGAuto);
END_IF;

@END_Body

@@@BEG_Comment@@@
@TL(0)

@@@END_Comment@@@

@BEG_SfcBody
16 13 17

@BEG_SfcData 2
@StepSeq @RT(4)sseq @F 3
@Step @RT(4)INIT @F @T @F @F @RT(0) @F
@AcbCont @RT(7)unnamed @F 1
@Acb @RT(5)aInit @F @F @RT(1)P @RT(0) @F @F @F @F

@Trans @RT(11)SimRequired @F @T @F @F @T @T @TL(2)
sv_bSimulate

@RT(7)Trans11 @F
@Loop @RT(4)loop @F 2
@StepSeq @RT(3)seq @F 3
@Step @RT(3)SIM @F @F @F @F @RT(0) @F
@AcbCont @RT(7)unnamed @F 1
@Acb @RT(9)aSimulate @F @F @RT(1)N @RT(0) @F @F @T @F

@Trans @RT(14)StpSimRequired @F @T @F @F @T @T @TL(2)
NOT sv_bSimulate

@RT(7)Trans13 @F
@Step @RT(4)STOP @F @F @F @F @RT(0) @F
@AcbCont @RT(7)unnamed @F 1
@Acb @RT(9)aStopSimu @F @F @RT(1)P @RT(0) @F @F @T @F

@Trans @RT(6)Return @F @T @T @T @T @T @TL(2)
TRUE

@RT(7)Trans16 @F

@END_SfcData
@SaActions 3
@SaText @RT(9)aSimulate 1 @TL(22)
(**************************************** WARNING ********************************************
 *** The KEBA Kemro K2 System including software is not intended for safety control tasks! ***
 ***                       For further information see Comment tab!                        ***
 *********************************************************************************************)

IF mFirstTimeRun THEN
   sv_ForceSGMoldClose := TRUE;
   sv_ForceSGNozzleClose := TRUE;
   sv_ForceSGNozzleRearClose := TRUE;
   sv_ForceSGRearClose := TRUE;
   sv_ForceEmergencyStop1 := TRUE;
   sv_ForceEmergencyStop2 := TRUE;
   sv_ForceEmergencyStop3 := TRUE;
   sv_ForceEmergencyStop4 := TRUE;
   sv_ForceOilFilterOK := FALSE;
   sv_ForceLightCurtainClose := TRUE;
   sv_ForceSafetyMat := TRUE;
   abForceMoldOpenMaxLimitSwitch.aSetForceValue(TRUE);
   abForceMoldCloseMinLimitSwitch.aSetForceValue(TRUE);
   mFirstTimeRun := FALSE;
END_IF;

@SaText @RT(9)aStopSimu 1 @TL(57)
IF mbDIEmergencyStop1Linked THEN
   fbEPUnForceDI(sSysVar := 'OperationMode1.di_EmergencyStop1');
END_IF;
IF mbDIEmergencyStop2Linked THEN
   fbEPUnForceDI(sSysVar := 'OperationMode1.di_EmergencyStop2');
END_IF;
IF mbDIEmergencyStop3Linked THEN
   fbEPUnForceDI(sSysVar := 'OperationMode1.di_EmergencyStop3');
END_IF;
IF mbDIEmergencyStop4Linked THEN
   fbEPUnForceDI(sSysVar := 'OperationMode1.di_EmergencyStop4');
END_IF;

IF mbDIOilFilterOkLinked THEN
   fbEPUnForceDI(sSysVar := 'OilMaintenance1.di_OilFilterOK');
END_IF;

// SG nozzle
IF mbDISGNozzleLinked THEN
   fbEPUnForceDI(sSysVar := 'SafetyGateNozzle1.di_Closed');
END_IF;

// SG nozzle rear
IF mbDISGNozzleRearLinked THEN
   fbEPUnForceDI(sSysVar := 'SafetyGateNozzleRear1.di_Closed');
END_IF;

// SG rear
IF mbDISGRearLinked THEN
   fbEPUnForceDI(sSysVar := 'SafetyGateRear1.di_Closed');
END_IF;

// SG mold
IF mbDISGMoldLinked THEN
   fbEPUnForceDI(sSysVar := 'SafetyGateMold1.di_Closed');
END_IF;
IF mbDISGMoldOpenLinked THEN
   fbEPUnForceDI(sSysVar := 'SafetyGateMold1.di_Open');
END_IF;

IF mbDISafetyMat1Linked THEN
   fbEPUnForceDI(sSysVar := 'SafetyMat1.di_SafetyMat');
END_IF;
IF mbDISafetyMat2Linked THEN
   fbEPUnForceDI(sSysVar := 'SafetyMat2.di_SafetyMat');
END_IF;

IF mbDILightCurtainClosedLinked THEN
   fbEPUnForceDI(sSysVar := 'LightCurtain1.di_Closed');
END_IF;

abForceMoldOpenMaxLimitSwitch.aUnforce();
abForceMoldCloseMinLimitSwitch.aUnforce();

mFirstTimeRun := TRUE;
STOP_PROCESS_ALGORITHM();

@SaText @RT(5)aInit 1 @TL(8)
(**************************************** WARNING ********************************************
 *** The KEBA Kemro K2 System including software is not intended for safety control tasks! ***
 ***                       For further information see Comment tab!                        ***
 *********************************************************************************************)

abForceMoldOpenMaxLimitSwitch.aInit('Mold1.di_MoldOpenProtect');
abForceMoldCloseMinLimitSwitch.aInit('Mold1.di_MoldCloseProtect');

@SaTrans 0
@SaExits 0
@END_SfcBody

@@@BEG_Comment@@@
@TL(0)

@@@END_Comment@@@

@BEG_Body
@TL(17)
IF sv_bSimulate THEN
   IF mbDIEmergencyStop1Linked THEN
      fbEPForceDI(sSysVar := 'OperationMode1.di_EmergencyStop1', Value := sv_ForceEmergencyStop1);
   END_IF;
   IF mbDIEmergencyStop2Linked THEN
      fbEPForceDI(sSysVar := 'OperationMode1.di_EmergencyStop2', Value := sv_ForceEmergencyStop2);
   END_IF;
   IF mbDIEmergencyStop3Linked THEN
      fbEPForceDI(sSysVar := 'OperationMode1.di_EmergencyStop3', Value := sv_ForceEmergencyStop3);
   END_IF;
   IF mbDIEmergencyStop4Linked THEN
      fbEPForceDI(sSysVar := 'OperationMode1.di_EmergencyStop4', Value := sv_ForceEmergencyStop4);
   END_IF;
END_IF;

@END_Body

@@@BEG_Comment@@@
@TL(0)

@@@END_Comment@@@

@BEG_Body
@TL(6)
IF mbDIOilFilterOkLinked THEN
   IF sv_bSimulate THEN
      fbEPForceDI(sSysVar := 'OilMaintenance1.di_OilFilterOK', Value := sv_ForceOilFilterOK);
   END_IF;
END_IF;

@END_Body

@@@BEG_Comment@@@
@TL(0)

@@@END_Comment@@@

@BEG_Body
@TL(10)
IF sv_bSimulate THEN
   IF mbDISGMoldLinked THEN
      fbEPForceDI(sSysVar :='SafetyGateMold1.di_Closed', Value := sv_ForceSGMoldClose);
   END_IF;
   IF mbDISGMoldOpenLinked THEN
      fbEPForceDI(sSysVar := 'SafetyGateMold1.di_Open', Value := NOT sv_ForceSGMoldClose);
   END_IF;
END_IF;

@END_Body

@@@BEG_Comment@@@
@TL(0)

@@@END_Comment@@@

@BEG_Body
@TL(7)
IF sv_bSimulate THEN
   IF mbDISGNozzleLinked THEN
      fbEPForceDI(sSysVar :='SafetyGateNozzle1.di_Closed', Value := sv_ForceSGNozzleClose);
   END_IF;
END_IF;

@END_Body

@@@BEG_Comment@@@
@TL(0)

@@@END_Comment@@@

@BEG_Body
@TL(7)
IF sv_bSimulate THEN
   IF mbDISGNozzleRearLinked THEN
      fbEPForceDI(sSysVar :='SafetyGateNozzleRear1.di_Closed', Value := sv_ForceSGNozzleRearClose);
   END_IF;
END_IF;

@END_Body

@@@BEG_Comment@@@
@TL(0)

@@@END_Comment@@@

@BEG_Body
@TL(7)
IF sv_bSimulate THEN
   IF mbDISGRearLinked THEN
      fbEPForceDI(sSysVar :='SafetyGateRear1.di_Closed', Value := sv_ForceSGRearClose);
   END_IF;
END_IF;

@END_Body

@@@BEG_Comment@@@
@TL(0)

@@@END_Comment@@@

@BEG_Body
@TL(7)
IF sv_bSimulate THEN
   IF mbDILightCurtainClosedLinked THEN
      fbEPForceDI(sSysVar :='LightCurtain1.di_Closed', Value := sv_ForceLightCurtainClose);
   END_IF;
END_IF;

@END_Body

@@@BEG_Comment@@@
@TL(0)

@@@END_Comment@@@

@BEG_Body
@TL(10)
IF sv_bSimulate THEN
   IF mbDISafetyMat1Linked THEN
      fbEPForceDI(sSysVar :='SafetyMat1.di_SafetyMat', Value := sv_ForceSafetyMat);
   END_IF;
   IF mbDISafetyMat2Linked THEN
      fbEPForceDI(sSysVar :='SafetyMat2.di_SafetyMat', Value := sv_ForceSafetyMat);
   END_IF;
END_IF;

@END_Body

@@@BEG_Comment@@@
@TL(0)

@@@END_Comment@@@

@BEG_Body
@TL(81)
pbDummy := GET_SYNC_REFTO('OperationMode1.di_EmergencyStop1', T#0s, Status);
mbDIEmergencyStop1Linked := (Status = KSYS_Status_OK);
pbDummy := GET_SYNC_REFTO('OperationMode1.di_EmergencyStop2', T#0s, Status);
mbDIEmergencyStop2Linked := (Status = KSYS_Status_OK);
pbDummy := GET_SYNC_REFTO('OperationMode1.di_EmergencyStop3', T#0s, Status);
mbDIEmergencyStop3Linked := (Status = KSYS_Status_OK);
pbDummy := GET_SYNC_REFTO('OperationMode1.di_EmergencyStop4', T#0s, Status);
mbDIEmergencyStop4Linked := (Status = KSYS_Status_OK);

pbDummy := GET_SYNC_REFTO('OilMaintenance1.di_OilFilterOK', T#0s, Status);
mbDIOilFilterOkLinked := (Status = KSYS_Status_OK);

pbDummy := GET_SYNC_REFTO('SafetyGateNozzle1.di_Closed', T#0s, Status);
mbDISGNozzleLinked := (Status = KSYS_Status_OK);

(*Optional Safety Gate Nozzle Rear*)
pbDummy := GET_SYNC_REFTO('SafetyGateNozzleRear1.di_Closed', T#0s, Status);
mbDISGNozzleRearLinked := (Status = KSYS_Status_OK);

// Safety Gate Rear
pbDummy := GET_SYNC_REFTO('SafetyGateRear1.di_Closed', T#0s, Status);
mbDISGRearLinked := (Status = KSYS_Status_OK);

// Safety Gate Mold
pbDummy := GET_SYNC_REFTO('SafetyGateMold1.di_Closed', T#0s, Status);
mbDISGMoldLinked := (Status = KSYS_Status_OK);
pbDummy := GET_SYNC_REFTO('SafetyGateMold1.di_Open', T#0s, Status);
mbDISGMoldOpenLinked := (Status = KSYS_Status_OK);

// SafetyGateAuto
mpbDISGAutoClosed1 := GET_SYNC_REFTO('SafetyGateAuto1.di_Closed', T#0s, Status);
mbDISGAutoClosed1Linked := (Status = KSYS_Status_OK);

mpbDISGAutoClosed2 := GET_SYNC_REFTO('SafetyGateAuto1.di_Closed2', T#0s, Status);
mbDISGAutoClosed2Linked := (Status = KSYS_Status_OK);

mpbDISGAutoOpen := GET_SYNC_REFTO('SafetyGateAuto1.di_Open', T#0s, Status);
mbDISGAutoOpenLinked := (Status = KSYS_Status_OK);

mpbDISGAutoCloseSlow := GET_SYNC_REFTO('SafetyGateAuto1.di_CloseSlow', T#0s, Status);
mbDISGAutoCloseSlowLinked := (Status = KSYS_Status_OK);

pbDummy := GET_SYNC_REFTO('SafetyGateAuto1.di_OpenSlow', T#0s, Status);
mbDISGAutoOpenSlowLinked := (Status = KSYS_Status_OK);

mpbDISGAutoLocked := GET_SYNC_REFTO('SafetyGateAuto1.di_Locked', T#0s, Status);
mbDISGAutoLockedLinked := (Status = KSYS_Status_OK);

mpbDISGAutoUnlocked := GET_SYNC_REFTO('SafetyGateAuto1.di_Unlocked', T#0s, Status);
mbDISGAutoUnlockedLinked := (Status = KSYS_Status_OK);

mpbDOSGAutoClose := GET_SYNC_REFTO('SafetyGateAuto1.do_Close', T#0s, Status);
mbDOSGAutoCloseLinked := (Status = KSYS_Status_OK);

mpbDOSGAutoFast := GET_SYNC_REFTO('SafetyGateAuto1.do_Fast', T#0s, Status);
mbDOSGAutoFastLinked := (Status = KSYS_Status_OK);

mpbDOSGAutoOpen := GET_SYNC_REFTO('SafetyGateAuto1.do_Open', T#0s, Status);
mbDOSGAutoOpenLinked := (Status = KSYS_Status_OK);

mpbDOSGAutoLock := GET_SYNC_REFTO('SafetyGateAuto1.do_Lock', T#0s, Status);
mbDOSGAutoLockLinked := (Status = KSYS_Status_OK);

mpbDOSGAutoUnlock := GET_SYNC_REFTO('SafetyGateAuto1.do_Unlock', T#0s, Status);
mbDOSGAutoUnlockLinked := (Status = KSYS_Status_OK);

// SafetyMat
pbDummy := GET_SYNC_REFTO('SafetyMat1.di_SafetyMat', T#0s, Status);
mbDISafetyMat1Linked := (Status = KSYS_Status_OK);

pbDummy := GET_SYNC_REFTO('SafetyMat2.di_SafetyMat', T#0s, Status);
mbDISafetyMat2Linked := (Status = KSYS_Status_OK);

//LightCurtain
pbDummy:= GET_SYNC_REFTO('LightCurtain1.di_Closed', T#0s, Status);
mbDILightCurtainClosedLinked := (Status = KSYS_Status_OK);

STOP_PROCESS_ALGORITHM();

@END_Body

@@@BEG_Comment@@@
@TL(0)

@@@END_Comment@@@

@BEG_SfcBody
2 2 1

@BEG_SfcData 2
@StepSeq @RT(4)sseq @F 3
@Step @RT(4)INIT @F @T @F @F @RT(0) @F
@AcbCont @RT(7)unnamed @F 0

@Trans @RT(11)SimRequired @F @T @F @F @T @T @TL(2)
sv_bSimulate

@RT(7)Trans11 @F
@Loop @RT(4)loop @F 2
@StepSeq @RT(3)seq @F 3
@Step @RT(3)SIM @F @F @F @F @RT(0) @F
@AcbCont @RT(7)unnamed @F 1
@Acb @RT(9)aSimulate @F @F @RT(1)N @RT(0) @F @F @T @F

@Trans @RT(14)StpSimRequired @F @T @F @F @T @T @TL(2)
NOT sv_bSimulate

@RT(7)Trans13 @F
@Step @RT(4)STOP @F @F @F @F @RT(0) @F
@AcbCont @RT(7)unnamed @F 1
@Acb @RT(9)aStopSimu @F @F @RT(1)P @RT(0) @F @F @T @F

@Trans @RT(6)Return @F @T @T @T @T @T @TL(2)
TRUE

@RT(7)Trans16 @F

@END_SfcData
@SaActions 2
@SaText @RT(9)aStopSimu 1 @TL(30)
IF mbDISGAutoClosed1Linked THEN
   fbEPUnForceDI(sSysVar := 'SafetyGateAuto1.di_Closed');
END_IF;

IF mbDISGAutoClosed2Linked THEN
   fbEPUnForceDI(sSysVar := 'SafetyGateAuto1.di_Closed2');
END_IF;

IF mbDISGAutoOpenLinked THEN
   fbEPUnForceDI(sSysVar := 'SafetyGateAuto1.di_Open');
END_IF;

IF mbDISGAutoOpenSlowLinked THEN
   fbEPUnForceDI(sSysVar := 'SafetyGateAuto1.di_OpenSlow');
END_IF;

IF mbDISGAutoCloseSlowLinked THEN
   fbEPUnForceDI(sSysVar := 'SafetyGateAuto1.di_CloseSlow');
END_IF;

IF mbDISGAutoLockedLinked THEN
   fbEPUnForceDI(sSysVar := 'SafetyGateAuto1.di_Locked');
END_IF;

IF mbDISGAutoUnlockedLinked THEN
   fbEPUnForceDI(sSysVar := 'SafetyGateAuto1.di_Unlocked');
END_IF;

STOP_PROCESS_ALGORITHM();

@SaText @RT(9)aSimulate 1 @TL(124)
//-------------------------------------------//
// normal movement simulation                //
//-------------------------------------------//

IF NOT bInitDone THEN
   fbEPForceDI(sSysVar := 'SafetyGateAuto1.di_Emergency',Value := TRUE);
   fbEPForceDI(sSysVar := 'SafetyGateAuto1.di_Emergency2',Value := TRUE);

   IF mbDISGAutoClosed1Linked THEN
      fbEPForceDI(sSysVar :='SafetyGateAuto1.di_Closed', Value := FALSE);
   END_IF;
   IF mbDISGAutoClosed2Linked THEN
      fbEPForceDI(sSysVar :='SafetyGateAuto1.di_Closed2', Value := TRUE);
   END_IF;
   IF mbDISGAutoCloseSlowLinked THEN
      fbEPForceDI(sSysVar :='SafetyGateAuto1.di_CloseSlow', Value := FALSE);
   END_IF;

   IF mbDISGAutoOpenLinked THEN
      fbEPForceDI(sSysVar :='SafetyGateAuto1.di_Open', Value := TRUE);
   END_IF;
   IF mbDISGAutoOpenSlowLinked THEN
      fbEPForceDI(sSysVar :='SafetyGateAuto1.di_OpenSlow', Value := TRUE);
   END_IF;

   IF mbDISGAutoLockedLinked THEN
      fbEPForceDI(sSysVar :='SafetyGateAuto1.di_Locked', Value := TRUE);
   END_IF;
   IF mbDISGAutoUnlockedLinked THEN
      fbEPForceDI(sSysVar :='SafetyGateAuto1.di_Unlocked', Value := FALSE);
   END_IF;

   bInitDone := TRUE;
END_IF;

// Safety Gate Close
IF mbDOSGAutoCloseLinked AND mpbDOSGAutoClose^ THEN

   IF mbDISGAutoOpenLinked AND mpbDISGAutoOpen^ THEN
      fbEPForceDI(sSysVar := 'SafetyGateAuto1.di_Open',Value := FALSE);
      fbEPForceDI(sSysVar := 'SafetyGateAuto1.di_OpenSlow',Value := FALSE);
   END_IF;

   IF mbDOSGAutoFastLinked THEN
       fbTimerSGAutoFast (IN := mpbDOSGAutoFast^,
                      PT := cTimeSGAutoFast);
   END_IF;
   IF fbTimerSGAutoFast.Q THEN
      fbTimerSGAutoFast(IN := FALSE);
      fbEPForceDI(sSysVar := 'SafetyGateAuto1.di_CloseSlow',Value := TRUE);
   END_IF;

   fbTimerSGAutoClose (IN := mpbDOSGAutoClose^,
                       PT := cTimeSGAutoClose);
   IF fbTimerSGAutoClose.Q THEN
      fbTimerSGAutoClose(IN := FALSE);
      fbEPForceDI(sSysVar := 'SafetyGateAuto1.di_Closed',Value := TRUE);
      fbEPForceDI(sSysVar := 'SafetyGateAuto1.di_Closed2',Value := FALSE);
   END_IF;
END_IF;

// Safety Gate Open
IF mbDOSGAutoOpenLinked AND mpbDOSGAutoOpen^ THEN
   IF mbDISGAutoClosed1Linked AND mpbDISGAutoClosed1^ THEN
      fbEPForceDI(sSysVar := 'SafetyGateAuto1.di_Closed',Value := FALSE);
      fbEPForceDI(sSysVar := 'SafetyGateAuto1.di_CloseSlow',Value := FALSE);
   END_IF;

   IF mbDISGAutoClosed2Linked AND NOT mpbDISGAutoClosed2^ THEN
      fbEPForceDI(sSysVar := 'SafetyGateAuto1.di_Closed2',Value := TRUE);
   END_IF;

   IF mbDOSGAutoFastLinked THEN
   fbTimerSGAutoFast (IN := mpbDOSGAutoFast^,
                      PT := cTimeSGAutoFast);
   END_IF;
   IF fbTimerSGAutoFast.Q THEN
      fbTimerSGAutoFast(IN := FALSE);
      fbEPForceDI(sSysVar := 'SafetyGateAuto1.di_OpenSlow',Value := TRUE);
   END_IF;

   fbTimerSGAutoOpen (IN := mpbDOSGAutoOpen^,
                       PT := cTimeSGAutoOpen);
   IF fbTimerSGAutoOpen.Q THEN
      fbTimerSGAutoOpen(IN := FALSE);
      fbEPForceDI(sSysVar := 'SafetyGateAuto1.di_Open',Value := TRUE);
   END_IF;
END_IF;

// Safety Gate Lock
IF mbDOSGAutoLockLinked AND mpbDOSGAutoLock^ THEN
   IF mbDISGAutoUnlockedLinked AND mpbDISGAutoUnlocked^ THEN
      fbEPForceDI(sSysVar := 'SafetyGateAuto1.di_Unlocked',Value := FALSE);
   END_IF;

   fbTimerSGAutoLock (IN := mpbDOSGAutoLock^,
                      PT := cTimeSGAutoLock);
   IF fbTimerSGAutoLock.Q THEN
      fbTimerSGAutoLock(IN := TRUE);
      fbEPForceDI(sSysVar := 'SafetyGateAuto1.di_Locked',Value := TRUE);
   END_IF;
END_IF;

// Safety Gate Unlock
IF mbDOSGAutoUnlockLinked AND mpbDOSGAutoUnlock^ THEN
   IF mbDISGAutoLockedLinked AND mpbDISGAutoLocked^ THEN
      fbEPForceDI(sSysVar := 'SafetyGateAuto1.di_Locked',Value := FALSE);
   END_IF;

   fbTimerSGAutoUnlock (IN := mpbDOSGAutoUnlock^,
                        PT := cTimeSGAutoUnlock);
   IF fbTimerSGAutoUnlock.Q THEN
      fbTimerSGAutoUnlock(IN := TRUE);
      fbEPForceDI(sSysVar := 'SafetyGateAuto1.di_Unlocked',Value := TRUE);
   END_IF;
END_IF;

@SaTrans 0
@SaExits 0
@END_SfcBody

@@@BEG_Comment@@@
@TL(0)

@@@END_Comment@@@
@END_Body

@END_Contents

(* ---- ABSpeedPumpSimu.pu ---- *)
IMPORT_OVER_LISTFILE
 GET_SYNC_REFTO
, cApplPlasticsPI
, KSYS_Status
, tOptionId
, KSWO_Status

END_IMPORT

ALGORITHM_BLOCK ABSpeedPumpSimu #DUMMY_EDIT_BLOCK

SYSTEM_VAR
 sv_bSimulate : BOOL;
 sv_bInitStart : BOOL;
END_VAR

SYSTEM_OBJECT
 TaskSim : TASK;
 TaskSlow : TASK;
 TaskInject : TASK;
 TaskAnalog : TASK;
 PU_Task_13 : TASK;
END_OBJECT

VAR
 mpMasterState : REFTO DWORD;
 mpSlave1State : REFTO DWORD;
 mpSlave2State : REFTO DWORD;
 mprSetPressureMaster : REFTO REAL;
 mprSetVelocityMaster : REFTO REAL;
 mprSetPressureSlave1 : REFTO REAL;
 mprSetVelocitySlave1 : REFTO REAL;
 mprSetPressureSlave2 : REFTO REAL;
 mprSetVelocitySlave2 : REFTO REAL;
 mbMotorOnReq : BOOL;
 mpbKeyOnOff : REFTO BOOL;
 mpbKeyOnOffHMI : REFTO BOOL;
 mpbMotorLocked : REFTO BOOL;
 mbSpeedPump : BOOL;
 mrAccelerationMaster : REAL;
 mrAccelerationSlave1 : REAL;
 mrAccelerationSlave2 : REAL;
 mprMotorPowerMaster : REFTO REAL;
 mprMotorPowerSlave1 : REFTO REAL;
 mprTorqueMaster : REFTO REAL;
 mprTorqueSlave1 : REFTO REAL;
 mpbInjectionActive : REFTO BOOL;
 mprActVelocitySlave1 : REFTO REAL;
 mprActVelocityMaster : REFTO REAL;
 mprActVelocitySlave2 : REFTO REAL;
 mpsRevisionMaster : REFTO STRING(255);
 mpsDrvIDMaster : REFTO STRING(255);
 mpiDriveStatusMaster : REFTO INT;
 mpsRevisionSlave1 : REFTO STRING(255);
 mpsDrvIDSlave1 : REFTO STRING(255);
 mpiDriveStatusSlave1 : REFTO INT;
 miCount : INT;
 mpiDriveStatusSlave2 : REFTO INT;
 mpsRevisionSlave2 : REFTO STRING(255);
 mpsDrvIDSlave2 : REFTO STRING(255);
 mprTorqueSlave2 : REFTO REAL;
 mprMotorPowerSlave2 : REFTO REAL;
 mbSlave1Linked : BOOL;
 mbSlave2Linked : BOOL;
END_VAR

PROCESS_ALGORITHM paSimulate ON TaskAnalog

VAR_TEMP
 b : BOOL;
END_VAR

VAR
 Status : KSYS_Status;
 rLastVelocityMaster : REAL;
 rLastVelocitySlave1 : REAL;
 rLastVelocitySlave2 : REAL;
 k1 : REAL := 0.1  (* Inertia (kg*m^2) *);
 k2 : REAL := 1.5 (* Coefficient (Nm/bar) *);
 k3 : REAL := 0.5 (* Friction coefficient (Nm/rad/s) *);
 rMaxVelocity : REAL := 209.44 (* rad/s *);
 dCycleTime : TIME;
 rCycleTime : REAL;
 rMaxPressure : REAL := 250.0 (* bar *);
 rLoadTorque : REAL := 1.0;
 sRevisionMaster : STRING(255) := 'AxX System Application V1-7-138';
 sDrvIDMaster : STRING(255) := 'AxM-II.35.70.4F';
 rActVelocityMaster : REAL;
 rActPressureMaster : REAL;
 rActVelocitySlave1 : REAL;
 rActPressureSlave1 : REAL;
 rActVelocitySlave2 : REAL;
 rActPressureSlave2 : REAL;
END_VAR

(* IecGraph-Code *)

(* init step *)
INITIAL_STEP INIT:
aInit (P);
END_STEP

(* steps *)
STEP SIM:
aReadDriveInfo (P);
aSimulate (N);
END_STEP

STEP STOP:
aStopSimu (P);
END_STEP

(* transitions *)
TRANSITION SimRequired (* SimRequired *) FROM INIT TO SIM :=  #BEGIN_EDIT_BLOCK
sv_bSimulate
;#END_EDIT_BLOCK
END_TRANSITION

TRANSITION StpSimRequired (* StpSimRequired *) FROM SIM TO STOP :=  #BEGIN_EDIT_BLOCK
NOT sv_bSimulate
;#END_EDIT_BLOCK
END_TRANSITION

TRANSITION Return (* Return *) FROM STOP TO SIM :=  #BEGIN_EDIT_BLOCK
TRUE
;#END_EDIT_BLOCK
END_TRANSITION

(* end IecGraph-Code *)
(* sfc-code *)

(* stand alone actions *)
ACTION aInit: #BEGIN_EDIT_BLOCK
(**************************************** WARNING ********************************************
 *** The KEBA Kemro K2 System including software is not intended for safety control tasks! ***
 ***                       For further information see Comment tab!                        ***
 *********************************************************************************************)
(*pointers*)
mpbKeyOnOff := GET_SYNC_REFTO("ServoDrives1.sv_KeyMotorOnOff", T#0s, Status);
// additionally listen to HMI on/off button (both can be linked)
mpbKeyOnOffHMI := GET_SYNC_REFTO("ServoDrives1.sv_KeyMotorOnOffHMI", T#0s, Status);

mpbMotorLocked := GET_SYNC_REFTO("ServoDrives1.sv_bMotorLocked", T#0s, Status);
mpbInjectionActive := GET_SYNC_REFTO("Injection1.sv_bInjectionActive", t#0s, Status);

(*Master*)
mprSetPressureMaster := GET_SYNC_REFTO('Pump1.sv_KHW_ServoMaster_setValue.rAux[1]', T#0s, Status);
mprSetVelocityMaster := GET_SYNC_REFTO('Pump1.sv_KHW_ServoMaster_setValue.rVeloc', T#0s, Status);
mprActVelocityMaster := GET_SYNC_REFTO("Pump1.sv_rActVelocityMaster", t#0s, Status);
mpMasterState := GET_SYNC_REFTO("Pump1.sv_KHW_ServoMaster_state_sim", T#0s, Status);
IF Status <> KSYS_Status_OK THEN
   mpMasterState := GET_SYNC_REFTO("Pump1.sv_KHW_ServoMaster_state", T#0s, Status);
END_IF;
mpiDriveStatusMaster := GET_SYNC_REFTO("Pump1.sv_iDriveStatusMaster", t#0s, Status);
mpsRevisionMaster := GET_SYNC_REFTO("Pump1.sv_sRevisionMaster", t#0s, Status);
mpsDrvIDMaster := GET_SYNC_REFTO("Pump1.sv_sDrvID_Master", t#0s, Status);
mprTorqueMaster := GET_SYNC_REFTO("Pump1.sv_rMotorTorqueMaster", T#0s, Status);
mprMotorPowerMaster := GET_SYNC_REFTO("Pump1.sv_rMotorPowerMaster", T#0s, Status);

(*Slave1*)
IF mbSlave1Linked THEN
   mprSetPressureSlave1 := GET_SYNC_REFTO('Pump1.sv_KHW_ServoSlave1_setValue.rAux[1]', T#0s, Status);
   mprSetVelocitySlave1 := GET_SYNC_REFTO('Pump1.sv_KHW_ServoSlave1_setValue.rVeloc', T#0s, Status);
   mpSlave1State := GET_SYNC_REFTO("Pump1.sv_KHW_ServoSlave1_state_sim", T#0s, Status);
   IF Status <> KSYS_Status_OK THEN
      mpSlave1State := GET_SYNC_REFTO("Pump1.sv_KHW_ServoSlave1_state", T#0s, Status);
   END_IF;
   mprActVelocitySlave1 := GET_SYNC_REFTO("Pump1.sv_rActVelocitySlave1", t#0s, Status);
   mpiDriveStatusSlave1 := GET_SYNC_REFTO("Pump1.sv_iDriveStatusSlave1", t#0s, Status);
   mpsRevisionSlave1 := GET_SYNC_REFTO("Pump1.sv_sRevisionSlave1", t#0s, Status);
   mpsDrvIDSlave1 := GET_SYNC_REFTO("Pump1.sv_sDrvID_Slave1", t#0s, Status);
   mprTorqueSlave1 := GET_SYNC_REFTO("Pump1.sv_rMotorTorqueSlave1", T#0s, Status);
   mprMotorPowerSlave1 := GET_SYNC_REFTO("Pump1.sv_rMotorPowerSlave1", T#0s, Status);
END_IF;

(*Slave2*)
IF mbSlave2Linked THEN
   mprSetPressureSlave2 := GET_SYNC_REFTO('Pump1.sv_KHW_ServoSlave2_setValue.rAux[1]', T#0s, Status);
   mprSetVelocitySlave2 := GET_SYNC_REFTO('Pump1.sv_KHW_ServoSlave2_setValue.rVeloc', T#0s, Status);
   mpSlave2State := GET_SYNC_REFTO("Pump1.sv_KHW_ServoSlave2_state_sim", T#0s, Status);
   IF Status <> KSYS_Status_OK THEN
      mpSlave2State := GET_SYNC_REFTO("Pump1.sv_KHW_ServoSlave2_state", T#0s, Status);
   END_IF;
   mprActVelocitySlave2 := GET_SYNC_REFTO("Pump1.sv_rActVelocitySlave2", t#0s, Status);
   mpiDriveStatusSlave2 := GET_SYNC_REFTO("Pump1.sv_iDriveStatusSlave2", t#0s, Status);
   mpsRevisionSlave2 := GET_SYNC_REFTO("Pump1.sv_sRevisionSlave2", t#0s, Status);
   mpsDrvIDSlave2:= GET_SYNC_REFTO("Pump1.sv_sDrvID_Slave2", t#0s, Status);
   mprTorqueSlave2 := GET_SYNC_REFTO("Pump1.sv_rMotorTorqueSlave2", T#0s, Status);
   mprMotorPowerSlave2 := GET_SYNC_REFTO("Pump1.sv_rMotorPowerSlave2", T#0s, Status);
END_IF;

dCycleTime := GET_TASK_INTERVAL();
rCycleTime := (LINT_TO_REAL(TIME_TO_LINT(dCycleTime))) / 1000000.0;

;#END_EDIT_BLOCK END_ACTION (*aInit*)
ACTION aStopSimu: #BEGIN_EDIT_BLOCK
(**************************************** WARNING ********************************************
 *** The KEBA Kemro K2 System including software is not intended for safety control tasks! ***
 ***                       For further information see Comment tab!                        ***
 *********************************************************************************************)

STOP_PROCESS_ALGORITHM();

;#END_EDIT_BLOCK END_ACTION (*aStopSimu*)
ACTION aSimulate: #BEGIN_EDIT_BLOCK
(**************************************** WARNING ********************************************
 *** The KEBA Kemro K2 System including software is not intended for safety control tasks! ***
 ***                       For further information see Comment tab!                        ***
 *********************************************************************************************)

(*Get the feedback directly from the set values in case of simulation mode*)
(*scaling : 1000% -> 100%*)
rActPressureMaster := mprSetPressureMaster^ / 10.0;
rActVelocityMaster := mprSetVelocityMaster^ / 10.0;
IF mbSlave1Linked THEN
   rActPressureSlave1 := mprSetPressureSlave1^ / 10.0;
   rActVelocitySlave1 := mprSetVelocitySlave1^ / 10.0;
END_IF;
IF mbSlave2Linked THEN
   rActPressureSlave2 := mprSetPressureSlave2^ / 10.0;
   rActVelocitySlave2 := mprSetVelocitySlave2^ / 10.0;
END_IF;

(*Velocity simulation*)
b := WRITE_SVREAL_DIRECT(mprActVelocityMaster^, (rMaxVelocity * rActVelocityMaster  / 100.0 * 30.0 / cApplPlasticsPI)); (*in rpm*)
IF mbSlave1Linked THEN
   b := WRITE_SVREAL_DIRECT(mprActVelocitySlave1^, (rMaxVelocity * rActVelocitySlave1  / 100.0 * 30.0 / cApplPlasticsPI)); (*in rpm*)
END_IF;
IF mbSlave2Linked THEN
   b := WRITE_SVREAL_DIRECT(mprActVelocitySlave2^, (rMaxVelocity * rActVelocitySlave2  / 100.0 * 30.0 / cApplPlasticsPI)); (*in rpm*)
END_IF;

(*Limitation of acceleration in simulation*)
IF rCycleTime <> 0.0 THEN
   mrAccelerationMaster := LIMIT(-14000.0, (rActVelocityMaster - rLastVelocityMaster) /100.0 * rMaxVelocity / rCycleTime, 14000.0);
   IF mbSlave1Linked THEN
      mrAccelerationSlave1 := LIMIT(-14000.0, (rActVelocitySlave1 - rLastVelocitySlave1) /100.0 * rMaxVelocity / rCycleTime, 14000.0);
   END_IF;
   IF mbSlave2Linked THEN
      mrAccelerationSlave2 := LIMIT(-14000.0, (rActVelocitySlave2 - rLastVelocitySlave2) /100.0 * rMaxVelocity / rCycleTime, 14000.0);
   END_IF;
END_IF;

(*100ms as cycle time for torque and power updating*)
IF miCount = 25 THEN
   (* simulate the motor torque *)
   IF mpbInjectionActive^ THEN
      (* pressure-proptional torque is simulated only during injection *)
      b := WRITE_SVREAL_DIRECT(mprTorqueMaster^, (k1 * mrAccelerationMaster + k2 * rActPressureMaster / 100.0 * rMaxPressure + k3 * rActVelocityMaster / 100.0 * rMaxVelocity + rLoadTorque));
      IF mbSlave1Linked THEN
         b := WRITE_SVREAL_DIRECT(mprTorqueSlave1^, (k1 * mrAccelerationSlave1 + k2 * rActPressureSlave1 / 100.0 * rMaxPressure + k3 * rActVelocitySlave1 / 100.0 * rMaxVelocity + rLoadTorque));
      END_IF;
      IF mbSlave2Linked THEN
         b := WRITE_SVREAL_DIRECT(mprTorqueSlave2^, (k1 * mrAccelerationSlave2 + k2 * rActPressureSlave2 / 100.0 * rMaxPressure + k3 * rActVelocitySlave2 / 100.0 * rMaxVelocity + rLoadTorque));
      END_IF;
   ELSE
      b := WRITE_SVREAL_DIRECT(mprTorqueMaster^, (k1 * mrAccelerationMaster + k3 * rActVelocityMaster / 100.0 * rMaxVelocity + rLoadTorque));
      IF mbSlave1Linked THEN
         b := WRITE_SVREAL_DIRECT(mprTorqueSlave1^, (k1 * mrAccelerationSlave1 + k3 * rActVelocitySlave1 / 100.0 * rMaxVelocity + rLoadTorque));
      END_IF;
      IF mbSlave2Linked THEN
         b := WRITE_SVREAL_DIRECT(mprTorqueSlave2^, (k1 * mrAccelerationSlave2 + k3 * rActVelocitySlave2 / 100.0 * rMaxVelocity + rLoadTorque));
      END_IF;
   END_IF;

   (* simulate motor power *)
   b := WRITE_SVREAL_DIRECT(mprMotorPowerMaster^, (mprTorqueMaster^ * rActVelocityMaster / 100.0 * rMaxVelocity / 1000.0));
   IF mbSlave1Linked THEN
      b := WRITE_SVREAL_DIRECT(mprMotorPowerSlave1^, (mprTorqueSlave1^ * rActVelocitySlave1 / 100.0 * rMaxVelocity / 1000.0));
   END_IF;
   IF mbSlave2Linked THEN
      b := WRITE_SVREAL_DIRECT(mprMotorPowerSlave2^, (mprTorqueSlave2^ * rActVelocitySlave2 / 100.0 * rMaxVelocity / 1000.0));
   END_IF;

   miCount := 0;
ELSE
   miCount := miCount + 1;
END_IF;

rLastVelocityMaster := rActVelocityMaster;
rLastVelocitySlave1 := rActVelocitySlave1;
rLastVelocitySlave2 := rActVelocitySlave2;

;#END_EDIT_BLOCK END_ACTION (*aSimulate*)
ACTION aReadDriveInfo: #BEGIN_EDIT_BLOCK
(**************************************** WARNING ********************************************
 *** The KEBA Kemro K2 System including software is not intended for safety control tasks! ***
 ***                       For further information see Comment tab!                        ***
 *********************************************************************************************)

b := WRITE_SV_DIRECT(mpsRevisionMaster^, sRevisionMaster);
b := WRITE_SV_DIRECT(mpsDrvIDMaster^, sDrvIDMaster);

IF mbSlave1Linked THEN
   b := WRITE_SV_DIRECT(mpsRevisionSlave1^, sRevisionMaster);
   b := WRITE_SV_DIRECT(mpsDrvIDSlave1^, sDrvIDMaster);
END_IF;

IF mbSlave2Linked THEN
   b := WRITE_SV_DIRECT(mpsRevisionSlave2^, sRevisionMaster);
   b := WRITE_SV_DIRECT(mpsDrvIDSlave2^, sDrvIDMaster);
END_IF;

;#END_EDIT_BLOCK END_ACTION (*aReadDriveInfo*)
(* end sfc-code *)

END_ALGORITHM

POSTUPDATE_ALGORITHM pStart ON TaskSim WITH sv_bSimulate,sv_bInitStart

VAR
 s : KSYS_Status;
 pOptions : REFTO tOptionId;
 bInitDone : BOOL;
END_VAR
#BEGIN_EDIT_BLOCK
(**************************************** WARNING ********************************************
 *** The KEBA Kemro K2 System including software is not intended for safety control tasks! ***
 ***                       For further information see Comment tab!                        ***
 *********************************************************************************************)

IF NOT bInitDone THEN
   (*Check if the speed pump exists, simulation will not be started in case of no speedpump*)
   pOptions := GET_SYNC_REFTO('Pump1.sv_Options', T#0s, s);
   mbSpeedPump := (s = KSYS_Status_OK) AND ((pOptions^ AND cSubOpSpeedpumpMaster) = cSubOpSpeedpumpMaster);

   IF ((pOptions^ AND cSubOpSpeedpumpSlave2) = cSubOpSpeedpumpSlave2) THEN
      mbSlave1Linked := TRUE;
      mbSlave2Linked := TRUE;
   ELSIF ((pOptions^ AND cSubOpSpeedpumpSlave1) = cSubOpSpeedpumpSlave1) THEN
      mbSlave1Linked := TRUE;
   END_IF;

   bInitDone := TRUE;
END_IF;

IF sv_bSimulate AND mbSpeedPump THEN
   START_PROCESS_ALGORITHM(paSimulate);
END_IF;

;#END_EDIT_BLOCK END_ALGORITHM

POSTUPDATE_ALGORITHM pOnOff ON PU_Task_13(1) WITH mpbKeyOnOff^,mpbKeyOnOffHMI^,mpbMotorLocked^

VAR
 iDriveStatus : INT;
 DriveState : DWORD;
 bOnOff : BOOL;
END_VAR
#BEGIN_EDIT_BLOCK
(**************************************** WARNING ********************************************
 *** The KEBA Kemro K2 System including software is not intended for safety control tasks! ***
 ***                       For further information see Comment tab!                        ***
 *********************************************************************************************)
IF mbSpeedPump THEN

   bOnOff := FALSE;

   IF mpbKeyOnOff <> EMPTY THEN
      bOnOff := mpbKeyOnOff^;
   END_IF;

   IF mpbKeyOnOffHMI <> EMPTY THEN
      bOnOff := bOnOff OR mpbKeyOnOffHMI^;
   END_IF;

   IF (bOnOff OR mpbMotorLocked^) THEN
      mbMotorOnReq := (NOT mbMotorOnReq) AND (NOT mpbMotorLocked^);
   END_IF;

   (*Force the status word when motor is shut on or off,
   so that the state handler works in simulation mode*)
   IF mbMotorOnReq THEN
      DriveState := 16#27;
      iDriveStatus := 2;
   ELSE
      DriveState := 0;
      iDriveStatus := 1;
   END_IF;

   mpMasterState^ := DriveState;
   mpiDriveStatusMaster^ := iDriveStatus;

   IF mbSlave1Linked THEN
      mpSlave1State^ := DriveState;
      mpiDriveStatusSlave1^ := iDriveStatus;
   END_IF;

   IF mbSlave2Linked THEN
      mpSlave2State^ := DriveState;
      mpiDriveStatusSlave2^ := iDriveStatus;
   END_IF;
END_IF;

;#END_EDIT_BLOCK END_ALGORITHM

PROCESS_ALGORITHM paInitDebugMeasurement ON TaskSlow AUTOSTART

VAR
 fuName : STRING(255);
 variableName : STRING(255);
 swoState : KSWO_Status;
END_VAR
#BEGIN_EDIT_BLOCK
(**************************************** WARNING ********************************************
 *** The KEBA Kemro K2 System including software is not intended for safety control tasks! ***
 ***                       For further information see Comment tab!                        ***
 *********************************************************************************************)

fuName := GET_MY_FU_NAME();
variableName := CONCAT(fuName,'.rTorque Nm');
swoState := KSWO_AddVariable( Task := TaskInject,
                              Name := variableName,
                              Variable := mprTorqueMaster^);

variableName := CONCAT(fuName,'.rAcc rad/s/s');
swoState := KSWO_AddVariable( Task := TaskInject,
                              Name := variableName,
                              Variable := mrAccelerationMaster);
STOP_PROCESS_ALGORITHM();

;#END_EDIT_BLOCK END_ALGORITHM

END_ALGORITHM_BLOCK

#END_OF_IEC_PART

@Puma @IecEditor 6 127 @Pou 25
@@@BEG_Comment@@@

@@@END_Comment@@@

@BEG_Contents

@BEG_Func
@RT(17)FuncTreeContainer
1
@Var @RT(14)GET_SYNC_REFTO @RT(0) @T @T @DERIVED 0 @F @RT(22)KEBA_STANDARD_FUNCTION @F
@T
@BEG_Attrib
0 @RT(0) @RT(0)
@END_Attrib
1 1 @F @F @F @F

@END_Func

@BEG_Const
@RT(18)ConstTreeContainer
1
@Var @RT(15)cApplPlasticsPI @RT(0) @T @F @DT @RT(4)REAL @RT(0) @T @T @BASIC 0 @F
@F @F
@T
@BEG_Attrib
0 @RT(10)3.14159265 @RT(13)pi=3.14159265
@END_Attrib
1 1 @F @F @F @F

@END_Const

@BEG_Export

@BEG_Kind
@ALGORITHM_BLOCK @RT(15)ABSpeedPumpSimu @STRUCTURED_TEXT
@RT(0) @RT(0) @RT(0)
@END_Kind

@BEG_Dcl
@RT(16)DclTreeContainer
46
@Var @RT(7)TaskSim @RT(0) @T @F @DT @RT(4)TASK @RT(0) @T @T @BASIC 0 @F
@F @F
@T
@BEG_Attrib
3 @RT(0) @RT(0) @RT(0)
@END_Attrib
1 7 @F @F @F @F

@Var @RT(8)TaskSlow @RT(0) @T @F @DT @RT(4)TASK @RT(0) @T @T @BASIC 0 @F
@F @F
@T
@BEG_Attrib
3 @RT(0) @RT(0) @RT(0)
@END_Attrib
1 7 @F @F @F @F

@Var @RT(10)TaskInject @RT(0) @T @F @DT @RT(4)TASK @RT(0) @T @T @BASIC 0 @F
@F @F
@T
@BEG_Attrib
3 @RT(0) @RT(0) @RT(0)
@END_Attrib
1 7 @F @F @F @F

@Var @RT(10)TaskAnalog @RT(0) @T @T @RENAMED 0 @T @T @DT @RT(4)TASK @RT(0) @T @T @BASIC 0 @F
@F @F
@T
@BEG_Attrib
3 @RT(0) @RT(0) @RT(0)
@END_Attrib
1 7 @F @F @F @F

@Var @RT(10)PU_Task_13 @RT(0) @T @F @DT @RT(4)TASK @RT(0) @T @T @BASIC 0 @F
@F @F
@T
@BEG_Attrib
3 @RT(0) @RT(0) @RT(0)
@END_Attrib
1 7 @F @F @F @F

@Var @RT(12)sv_bSimulate @RT(0) @T @F @DT @RT(4)BOOL @RT(0) @T @T @BASIC 0 @F
@F @F
@T
@BEG_Attrib
3 @RT(0) @RT(0) @RT(0)
@END_Attrib
1 8 @F @F @F @F

@Var @RT(13)sv_bInitStart @RT(0) @T @F @DT @RT(4)BOOL @RT(0) @T @T @BASIC 0 @F
@F @F
@T
@BEG_Attrib
3 @RT(0) @RT(0) @RT(0)
@END_Attrib
1 8 @F @F @F @F

@Var @RT(13)mpMasterState @RT(0) @T @T @REFTO 0 @T @DT @RT(5)DWORD @RT(0) @T @T @BASIC 0 @F
@F @F
@T
@BEG_Attrib
3 @RT(0) @RT(0) @RT(0)
@END_Attrib
1 0 @F @F @F @F

@Var @RT(13)mpSlave1State @RT(0) @T @T @REFTO 0 @T @DT @RT(5)DWORD @RT(0) @T @T @BASIC 0 @F
@F @F
@T
@BEG_Attrib
3 @RT(0) @RT(0) @RT(0)
@END_Attrib
1 0 @F @F @F @F

@Var @RT(13)mpSlave2State @RT(0) @T @T @REFTO 0 @T @DT @RT(5)DWORD @RT(0) @T @T @BASIC 0 @F
@F @F
@T
@BEG_Attrib
3 @RT(0) @RT(0) @RT(0)
@END_Attrib
1 0 @F @F @F @F

@Var @RT(20)mprSetPressureMaster @RT(0) @T @T @REFTO 0 @T @DT @RT(4)REAL @RT(0) @T @T @BASIC 0 @F
@F @F
@T
@BEG_Attrib
3 @RT(0) @RT(0) @RT(0)
@END_Attrib
1 0 @F @F @F @F

@Var @RT(20)mprSetVelocityMaster @RT(0) @T @T @REFTO 0 @T @DT @RT(4)REAL @RT(0) @T @T @BASIC 0 @F
@F @F
@T
@BEG_Attrib
3 @RT(0) @RT(0) @RT(0)
@END_Attrib
1 0 @F @F @F @F

@Var @RT(20)mprSetPressureSlave1 @RT(0) @T @T @REFTO 0 @T @DT @RT(4)REAL @RT(0) @T @T @BASIC 0 @F
@F @F
@T
@BEG_Attrib
3 @RT(0) @RT(0) @RT(0)
@END_Attrib
1 0 @F @F @F @F

@Var @RT(20)mprSetVelocitySlave1 @RT(0) @T @T @REFTO 0 @T @DT @RT(4)REAL @RT(0) @T @T @BASIC 0 @F
@F @F
@T
@BEG_Attrib
3 @RT(0) @RT(0) @RT(0)
@END_Attrib
1 0 @F @F @F @F

@Var @RT(20)mprSetPressureSlave2 @RT(0) @T @T @REFTO 0 @T @DT @RT(4)REAL @RT(0) @T @T @BASIC 0 @F
@F @F
@T
@BEG_Attrib
3 @RT(0) @RT(0) @RT(0)
@END_Attrib
1 0 @F @F @F @F

@Var @RT(20)mprSetVelocitySlave2 @RT(0) @T @T @REFTO 0 @T @DT @RT(4)REAL @RT(0) @T @T @BASIC 0 @F
@F @F
@T
@BEG_Attrib
3 @RT(0) @RT(0) @RT(0)
@END_Attrib
1 0 @F @F @F @F

@Var @RT(12)mbMotorOnReq @RT(0) @T @F @DT @RT(4)BOOL @RT(0) @T @T @BASIC 0 @F
@F @F
@T
@BEG_Attrib
3 @RT(0) @RT(0) @RT(0)
@END_Attrib
1 0 @F @F @F @F

@Var @RT(11)mpbKeyOnOff @RT(0) @T @T @REFTO 0 @T @DT @RT(4)BOOL @RT(0) @T @T @BASIC 0 @F
@F @F
@T
@BEG_Attrib
3 @RT(0) @RT(0) @RT(0)
@END_Attrib
1 0 @F @F @F @F

@Var @RT(14)mpbKeyOnOffHMI @RT(0) @T @T @REFTO 0 @T @DT @RT(4)BOOL @RT(0) @T @T @BASIC 0 @F
@F @F
@T
@BEG_Attrib
3 @RT(0) @RT(0) @RT(0)
@END_Attrib
1 0 @F @F @F @F

@Var @RT(14)mpbMotorLocked @RT(0) @T @T @REFTO 0 @T @DT @RT(4)BOOL @RT(0) @T @T @BASIC 0 @F
@F @F
@T
@BEG_Attrib
3 @RT(0) @RT(0) @RT(0)
@END_Attrib
1 0 @F @F @F @F

@Var @RT(11)mbSpeedPump @RT(0) @T @F @DT @RT(4)BOOL @RT(0) @T @T @BASIC 0 @F
@F @F
@T
@BEG_Attrib
3 @RT(0) @RT(0) @RT(0)
@END_Attrib
1 0 @F @F @F @F

@Var @RT(20)mrAccelerationMaster @RT(0) @T @F @DT @RT(4)REAL @RT(0) @T @T @BASIC 0 @F
@F @F
@T
@BEG_Attrib
3 @RT(0) @RT(0) @RT(0)
@END_Attrib
1 0 @F @F @F @F

@Var @RT(20)mrAccelerationSlave1 @RT(0) @T @F @DT @RT(4)REAL @RT(0) @T @T @BASIC 0 @F
@F @F
@T
@BEG_Attrib
3 @RT(0) @RT(0) @RT(0)
@END_Attrib
1 0 @F @F @F @F

@Var @RT(20)mrAccelerationSlave2 @RT(0) @T @F @DT @RT(4)REAL @RT(0) @T @T @BASIC 0 @F
@F @F
@T
@BEG_Attrib
3 @RT(0) @RT(0) @RT(0)
@END_Attrib
1 0 @F @F @F @F

@Var @RT(19)mprMotorPowerMaster @RT(0) @T @T @REFTO 0 @T @DT @RT(4)REAL @RT(0) @T @T @BASIC 0 @F
@F @F
@T
@BEG_Attrib
3 @RT(0) @RT(0) @RT(0)
@END_Attrib
1 0 @F @F @F @F

@Var @RT(19)mprMotorPowerSlave1 @RT(0) @T @T @REFTO 0 @T @DT @RT(4)REAL @RT(0) @T @T @BASIC 0 @F
@F @F
@T
@BEG_Attrib
3 @RT(0) @RT(0) @RT(0)
@END_Attrib
1 0 @F @F @F @F

@Var @RT(15)mprTorqueMaster @RT(0) @T @T @REFTO 0 @T @DT @RT(4)REAL @RT(0) @T @T @BASIC 0 @F
@F @F
@T
@BEG_Attrib
3 @RT(0) @RT(0) @RT(0)
@END_Attrib
1 0 @F @F @F @F

@Var @RT(15)mprTorqueSlave1 @RT(0) @T @T @REFTO 0 @T @DT @RT(4)REAL @RT(0) @T @T @BASIC 0 @F
@F @F
@T
@BEG_Attrib
3 @RT(0) @RT(0) @RT(0)
@END_Attrib
1 0 @F @F @F @F

@Var @RT(18)mpbInjectionActive @RT(0) @T @T @REFTO 0 @T @DT @RT(4)BOOL @RT(0) @T @T @BASIC 0 @F
@F @F
@T
@BEG_Attrib
3 @RT(0) @RT(0) @RT(0)
@END_Attrib
1 0 @F @F @F @F

@Var @RT(20)mprActVelocitySlave1 @RT(0) @T @T @REFTO 0 @T @DT @RT(4)REAL @RT(0) @T @T @BASIC 0 @F
@F @F
@T
@BEG_Attrib
3 @RT(0) @RT(0) @RT(0)
@END_Attrib
1 0 @F @F @F @F

@Var @RT(20)mprActVelocityMaster @RT(0) @T @T @REFTO 0 @T @DT @RT(4)REAL @RT(0) @T @T @BASIC 0 @F
@F @F
@T
@BEG_Attrib
3 @RT(0) @RT(0) @RT(0)
@END_Attrib
1 0 @F @F @F @F

@Var @RT(20)mprActVelocitySlave2 @RT(0) @T @T @REFTO 0 @T @DT @RT(4)REAL @RT(0) @T @T @BASIC 0 @F
@F @F
@T
@BEG_Attrib
3 @RT(0) @RT(0) @RT(0)
@END_Attrib
1 0 @F @F @F @F

@Var @RT(17)mpsRevisionMaster @RT(0) @T @T @REFTO 0 @T @DT @RT(11)STRING(255) @RT(0) @T @T @STRING 0 @F @RT(3)255 @F
@F @F
@T
@BEG_Attrib
3 @RT(0) @RT(0) @RT(0)
@END_Attrib
1 0 @F @F @F @F

@Var @RT(14)mpsDrvIDMaster @RT(0) @T @T @REFTO 0 @T @DT @RT(11)STRING(255) @RT(0) @T @T @STRING 0 @F @RT(3)255 @F
@F @F
@T
@BEG_Attrib
3 @RT(0) @RT(0) @RT(0)
@END_Attrib
1 0 @F @F @F @F

@Var @RT(20)mpiDriveStatusMaster @RT(0) @T @T @REFTO 0 @T @DT @RT(3)INT @RT(0) @T @T @BASIC 0 @F
@F @F
@T
@BEG_Attrib
3 @RT(0) @RT(0) @RT(0)
@END_Attrib
1 0 @F @F @F @F

@Var @RT(17)mpsRevisionSlave1 @RT(0) @T @T @REFTO 0 @T @DT @RT(11)STRING(255) @RT(0) @T @T @STRING 0 @F @RT(3)255 @F
@F @F
@T
@BEG_Attrib
3 @RT(0) @RT(0) @RT(0)
@END_Attrib
1 0 @F @F @F @F

@Var @RT(14)mpsDrvIDSlave1 @RT(0) @T @T @REFTO 0 @T @DT @RT(11)STRING(255) @RT(0) @T @T @STRING 0 @F @RT(3)255 @F
@F @F
@T
@BEG_Attrib
3 @RT(0) @RT(0) @RT(0)
@END_Attrib
1 0 @F @F @F @F

@Var @RT(20)mpiDriveStatusSlave1 @RT(0) @T @T @REFTO 0 @T @DT @RT(3)INT @RT(0) @T @T @BASIC 0 @F
@F @F
@T
@BEG_Attrib
3 @RT(0) @RT(0) @RT(0)
@END_Attrib
1 0 @F @F @F @F

@Var @RT(7)miCount @RT(0) @T @F @DT @RT(3)INT @RT(0) @T @T @BASIC 0 @F
@F @F
@T
@BEG_Attrib
3 @RT(0) @RT(0) @RT(0)
@END_Attrib
1 0 @F @F @F @F

@Var @RT(20)mpiDriveStatusSlave2 @RT(0) @T @T @REFTO 0 @T @DT @RT(3)INT @RT(0) @T @T @BASIC 0 @F
@F @F
@T
@BEG_Attrib
3 @RT(0) @RT(0) @RT(0)
@END_Attrib
1 0 @F @F @F @F

@Var @RT(17)mpsRevisionSlave2 @RT(0) @T @T @REFTO 0 @T @DT @RT(11)STRING(255) @RT(0) @T @T @STRING 0 @F @RT(3)255 @F
@F @F
@T
@BEG_Attrib
3 @RT(0) @RT(0) @RT(0)
@END_Attrib
1 0 @F @F @F @F

@Var @RT(14)mpsDrvIDSlave2 @RT(0) @T @T @REFTO 0 @T @DT @RT(11)STRING(255) @RT(0) @T @T @STRING 0 @F @RT(3)255 @F
@F @F
@T
@BEG_Attrib
3 @RT(0) @RT(0) @RT(0)
@END_Attrib
1 0 @F @F @F @F

@Var @RT(15)mprTorqueSlave2 @RT(0) @T @T @REFTO 0 @T @DT @RT(4)REAL @RT(0) @T @T @BASIC 0 @F
@F @F
@T
@BEG_Attrib
3 @RT(0) @RT(0) @RT(0)
@END_Attrib
1 0 @F @F @F @F

@Var @RT(19)mprMotorPowerSlave2 @RT(0) @T @T @REFTO 0 @T @DT @RT(4)REAL @RT(0) @T @T @BASIC 0 @F
@F @F
@T
@BEG_Attrib
3 @RT(0) @RT(0) @RT(0)
@END_Attrib
1 0 @F @F @F @F

@Var @RT(14)mbSlave1Linked @RT(0) @T @F @DT @RT(4)BOOL @RT(0) @T @T @BASIC 0 @F
@F @F
@T
@BEG_Attrib
3 @RT(0) @RT(0) @RT(0)
@END_Attrib
1 0 @F @F @F @F

@Var @RT(14)mbSlave2Linked @RT(0) @T @F @DT @RT(4)BOOL @RT(0) @T @T @BASIC 0 @F
@F @F
@T
@BEG_Attrib
3 @RT(0) @RT(0) @RT(0)
@END_Attrib
1 0 @F @F @F @F

@END_Dcl

@END_Export

@BEG_Body

4

@BEG_Export

@BEG_Algo
@PROCESS_ALGORITHM @RT(10)paSimulate @SEQUENTIAL_FLOW_CHART
@RT(0) @RT(0) @RT(10)TaskAnalog @F @F
@END_Algo

@BEG_Dcl
@RT(16)DclTreeContainer
21
@Var @RT(6)Status @RT(0) @T @T @DERIVED 0 @T @T @DT @RT(11)KSYS_Status @RT(0) @T @T @UNKNOWN 0 @F
@F @F
@T
@BEG_Attrib
3 @RT(0) @RT(0) @RT(0)
@END_Attrib
1 0 @F @F @F @F

@Var @RT(19)rLastVelocityMaster @RT(0) @T @F @DT @RT(4)REAL @RT(0) @T @T @BASIC 0 @F
@F @F
@T
@BEG_Attrib
3 @RT(0) @RT(0) @RT(0)
@END_Attrib
1 0 @F @F @F @F

@Var @RT(19)rLastVelocitySlave1 @RT(0) @T @F @DT @RT(4)REAL @RT(0) @T @T @BASIC 0 @F
@F @F
@T
@BEG_Attrib
3 @RT(0) @RT(0) @RT(0)
@END_Attrib
1 0 @F @F @F @F

@Var @RT(19)rLastVelocitySlave2 @RT(0) @T @F @DT @RT(4)REAL @RT(0) @T @T @BASIC 0 @F
@F @F
@T
@BEG_Attrib
3 @RT(0) @RT(0) @RT(0)
@END_Attrib
1 0 @F @F @F @F

@Var @RT(2)k1 @RT(0) @T @T @RENAMED 0 @T @T @DT @RT(4)REAL @RT(0) @T @T @BASIC 0 @F
@F @F
@T
@BEG_Attrib
3 @RT(4)0.1  @RT(16)Inertia (kg*m^2) @RT(0)
@END_Attrib
1 0 @F @F @F @F

@Var @RT(2)k2 @RT(0) @T @T @RENAMED 0 @T @T @DT @RT(4)REAL @RT(0) @T @T @BASIC 0 @F
@F @F
@T
@BEG_Attrib
3 @RT(3)1.5 @RT(20)Coefficient (Nm/bar) @RT(0)
@END_Attrib
1 0 @F @F @F @F

@Var @RT(2)k3 @RT(0) @T @T @RENAMED 0 @T @T @DT @RT(4)REAL @RT(0) @T @T @BASIC 0 @F
@F @F
@T
@BEG_Attrib
3 @RT(3)0.5 @RT(31)Friction coefficient (Nm/rad/s) @RT(0)
@END_Attrib
1 0 @F @F @F @F

@Var @RT(12)rMaxVelocity @RT(0) @T @F @DT @RT(4)REAL @RT(0) @T @T @BASIC 0 @F
@F @F
@T
@BEG_Attrib
3 @RT(6)209.44 @RT(5)rad/s @RT(0)
@END_Attrib
1 0 @F @F @F @F

@Var @RT(10)dCycleTime @RT(0) @T @T @RENAMED 0 @T @T @DT @RT(4)TIME @RT(0) @T @T @BASIC 0 @F
@F @F
@T
@BEG_Attrib
3 @RT(0) @RT(0) @RT(0)
@END_Attrib
1 0 @F @F @F @F

@Var @RT(10)rCycleTime @RT(0) @T @F @DT @RT(4)REAL @RT(0) @T @T @BASIC 0 @F
@F @F
@T
@BEG_Attrib
3 @RT(0) @RT(0) @RT(0)
@END_Attrib
1 0 @F @F @F @F

@Var @RT(12)rMaxPressure @RT(0) @T @F @DT @RT(4)REAL @RT(0) @T @T @BASIC 0 @F
@F @F
@T
@BEG_Attrib
3 @RT(5)250.0 @RT(3)bar @RT(0)
@END_Attrib
1 0 @F @F @F @F

@Var @RT(11)rLoadTorque @RT(0) @T @F @DT @RT(4)REAL @RT(0) @T @T @BASIC 0 @F
@F @F
@T
@BEG_Attrib
3 @RT(3)1.0 @RT(0) @RT(0)
@END_Attrib
1 0 @F @F @F @F

@Var @RT(15)sRevisionMaster @RT(0) @T @F @DT @RT(11)STRING(255) @RT(0) @T @T @STRING 0 @F @RT(3)255 @F
@F @F
@T
@BEG_Attrib
3 @RT(33)'AxX System Application V1-7-138' @RT(0) @RT(0)
@END_Attrib
1 0 @F @F @F @F

@Var @RT(12)sDrvIDMaster @RT(0) @T @F @DT @RT(11)STRING(255) @RT(0) @T @T @STRING 0 @F @RT(3)255 @F
@F @F
@T
@BEG_Attrib
3 @RT(17)'AxM-II.35.70.4F' @RT(0) @RT(0)
@END_Attrib
1 0 @F @F @F @F

@Var @RT(18)rActVelocityMaster @RT(0) @T @F @DT @RT(4)REAL @RT(0) @T @T @BASIC 0 @F
@F @F
@T
@BEG_Attrib
3 @RT(0) @RT(0) @RT(0)
@END_Attrib
1 0 @F @F @F @F

@Var @RT(18)rActPressureMaster @RT(0) @T @T @RENAMED 0 @T @T @DT @RT(4)REAL @RT(0) @T @T @BASIC 0 @F
@F @F
@T
@BEG_Attrib
3 @RT(0) @RT(0) @RT(0)
@END_Attrib
1 0 @F @F @F @F

@Var @RT(18)rActVelocitySlave1 @RT(0) @T @F @DT @RT(4)REAL @RT(0) @T @T @BASIC 0 @F
@F @F
@T
@BEG_Attrib
3 @RT(0) @RT(0) @RT(0)
@END_Attrib
1 0 @F @F @F @F

@Var @RT(18)rActPressureSlave1 @RT(0) @T @T @RENAMED 0 @T @T @DT @RT(4)REAL @RT(0) @T @T @BASIC 0 @F
@F @F
@T
@BEG_Attrib
3 @RT(0) @RT(0) @RT(0)
@END_Attrib
1 0 @F @F @F @F

@Var @RT(18)rActVelocitySlave2 @RT(0) @T @F @DT @RT(4)REAL @RT(0) @T @T @BASIC 0 @F
@F @F
@T
@BEG_Attrib
3 @RT(0) @RT(0) @RT(0)
@END_Attrib
1 0 @F @F @F @F

@Var @RT(18)rActPressureSlave2 @RT(0) @T @T @RENAMED 0 @T @T @DT @RT(4)REAL @RT(0) @T @T @BASIC 0 @F
@F @F
@T
@BEG_Attrib
3 @RT(0) @RT(0) @RT(0)
@END_Attrib
1 0 @F @F @F @F

@Var @RT(1)b @RT(0) @T @F @DT @RT(4)BOOL @RT(0) @T @T @BASIC 0 @F
@F @F
@T
@BEG_Attrib
3 @RT(0) @RT(0) @RT(0)
@END_Attrib
1 4 @F @F @F @F

@END_Dcl

@END_Export

@BEG_Export

@BEG_Algo
@POSTUPDATE_ALGORITHM @RT(6)pStart @STRUCTURED_TEXT
@RT(0) @RT(26)sv_bSimulate,sv_bInitStart @RT(7)TaskSim @F @F
@END_Algo

@BEG_Dcl
@RT(16)DclTreeContainer
3
@Var @RT(1)s @RT(0) @T @T @DERIVED 0 @T @T @DT @RT(11)KSYS_Status @RT(0) @T @T @UNKNOWN 0 @F
@F @F
@T
@BEG_Attrib
3 @RT(0) @RT(0) @RT(0)
@END_Attrib
1 0 @F @F @F @F

@Var @RT(8)pOptions @RT(0) @T @T @REFTO 0 @F @DERIVED 0 @T @T @DT @RT(9)tOptionId @RT(0) @T @T @UNKNOWN 0 @F
@F @F
@T
@BEG_Attrib
3 @RT(0) @RT(0) @RT(0)
@END_Attrib
1 0 @F @F @F @F

@Var @RT(9)bInitDone @RT(0) @T @F @DT @RT(4)BOOL @RT(0) @T @T @BASIC 0 @F
@F @F
@T
@BEG_Attrib
3 @RT(0) @RT(0) @RT(0)
@END_Attrib
1 0 @F @F @F @F

@END_Dcl

@END_Export

@BEG_Export

@BEG_Algo
@POSTUPDATE_ALGORITHM @RT(6)pOnOff @STRUCTURED_TEXT
@RT(0) @RT(44)mpbKeyOnOff^,mpbKeyOnOffHMI^,mpbMotorLocked^ @RT(13)PU_Task_13(1) @F @F
@END_Algo

@BEG_Dcl
@RT(16)DclTreeContainer
3
@Var @RT(12)iDriveStatus @RT(0) @T @F @DT @RT(3)INT @RT(0) @T @T @BASIC 0 @F
@F @F
@T
@BEG_Attrib
3 @RT(0) @RT(0) @RT(0)
@END_Attrib
1 0 @F @F @F @F

@Var @RT(10)DriveState @RT(0) @T @F @DT @RT(5)DWORD @RT(0) @T @T @BASIC 0 @F
@F @F
@T
@BEG_Attrib
3 @RT(0) @RT(0) @RT(0)
@END_Attrib
1 0 @F @F @F @F

@Var @RT(6)bOnOff @RT(0) @T @F @DT @RT(4)BOOL @RT(0) @T @T @BASIC 0 @F
@F @F
@T
@BEG_Attrib
3 @RT(0) @RT(0) @RT(0)
@END_Attrib
1 0 @F @F @F @F

@END_Dcl

@END_Export

@BEG_Export

@BEG_Algo
@PROCESS_ALGORITHM @RT(22)paInitDebugMeasurement @STRUCTURED_TEXT
@RT(0) @RT(0) @RT(8)TaskSlow @T @F
@END_Algo

@BEG_Dcl
@RT(16)DclTreeContainer
3
@Var @RT(6)fuName @RT(0) @T @F @DT @RT(11)STRING(255) @RT(0) @T @T @STRING 0 @F @RT(3)255 @F
@F @F
@T
@BEG_Attrib
3 @RT(0) @RT(0) @RT(0)
@END_Attrib
1 0 @F @F @F @F

@Var @RT(12)variableName @RT(0) @T @F @DT @RT(11)STRING(255) @RT(0) @T @T @STRING 0 @F @RT(3)255 @F
@F @F
@T
@BEG_Attrib
3 @RT(0) @RT(0) @RT(0)
@END_Attrib
1 0 @F @F @F @F

@Var @RT(8)swoState @RT(0) @T @T @DERIVED 0 @T @T @DT @RT(11)KSWO_Status @RT(0) @T @T @UNKNOWN 0 @F
@F @F
@T
@BEG_Attrib
3 @RT(0) @RT(0) @RT(0)
@END_Attrib
1 0 @F @F @F @F

@END_Dcl

@END_Export

@BEG_SfcBody
4 3 2

@BEG_SfcData 2
@StepSeq @RT(4)sseq @F 3
@Step @RT(4)INIT @F @T @F @F @RT(0) @F
@AcbCont @RT(7)unnamed @F 1
@Acb @RT(5)aInit @F @F @RT(1)P @RT(0) @F @F @F @F

@Trans @RT(11)SimRequired @F @T @F @F @T @T @TL(2)
sv_bSimulate

@RT(11)SimRequired @F
@Loop @RT(4)loop @F 2
@StepSeq @RT(4)sseq @F 3
@Step @RT(3)SIM @F @F @F @F @RT(0) @F
@AcbCont @RT(7)unnamed @F 2
@Acb @RT(14)aReadDriveInfo @F @F @RT(1)P @RT(0) @F @F @F @F
@Acb @RT(9)aSimulate @F @F @RT(1)N @RT(0) @F @F @F @F

@Trans @RT(14)StpSimRequired @F @T @F @F @T @T @TL(2)
NOT sv_bSimulate

@RT(14)StpSimRequired @F
@Step @RT(4)STOP @F @F @F @F @RT(0) @F
@AcbCont @RT(7)unnamed @F 1
@Acb @RT(9)aStopSimu @F @F @RT(1)P @RT(0) @F @F @F @F

@Trans @RT(6)Return @F @T @T @T @T @T @TL(2)
TRUE

@RT(6)Return @F

@END_SfcData
@SaActions 4
@SaText @RT(5)aInit 1 @TL(61)
(**************************************** WARNING ********************************************
 *** The KEBA Kemro K2 System including software is not intended for safety control tasks! ***
 ***                       For further information see Comment tab!                        ***
 *********************************************************************************************)
(*pointers*)
mpbKeyOnOff := GET_SYNC_REFTO("ServoDrives1.sv_KeyMotorOnOff", T#0s, Status);
// additionally listen to HMI on/off button (both can be linked)
mpbKeyOnOffHMI := GET_SYNC_REFTO("ServoDrives1.sv_KeyMotorOnOffHMI", T#0s, Status);

mpbMotorLocked := GET_SYNC_REFTO("ServoDrives1.sv_bMotorLocked", T#0s, Status);
mpbInjectionActive := GET_SYNC_REFTO("Injection1.sv_bInjectionActive", t#0s, Status);

(*Master*)
mprSetPressureMaster := GET_SYNC_REFTO('Pump1.sv_KHW_ServoMaster_setValue.rAux[1]', T#0s, Status);
mprSetVelocityMaster := GET_SYNC_REFTO('Pump1.sv_KHW_ServoMaster_setValue.rVeloc', T#0s, Status);
mprActVelocityMaster := GET_SYNC_REFTO("Pump1.sv_rActVelocityMaster", t#0s, Status);
mpMasterState := GET_SYNC_REFTO("Pump1.sv_KHW_ServoMaster_state_sim", T#0s, Status);
IF Status <> KSYS_Status_OK THEN
   mpMasterState := GET_SYNC_REFTO("Pump1.sv_KHW_ServoMaster_state", T#0s, Status);
END_IF;
mpiDriveStatusMaster := GET_SYNC_REFTO("Pump1.sv_iDriveStatusMaster", t#0s, Status);
mpsRevisionMaster := GET_SYNC_REFTO("Pump1.sv_sRevisionMaster", t#0s, Status);
mpsDrvIDMaster := GET_SYNC_REFTO("Pump1.sv_sDrvID_Master", t#0s, Status);
mprTorqueMaster := GET_SYNC_REFTO("Pump1.sv_rMotorTorqueMaster", T#0s, Status);
mprMotorPowerMaster := GET_SYNC_REFTO("Pump1.sv_rMotorPowerMaster", T#0s, Status);

(*Slave1*)
IF mbSlave1Linked THEN
   mprSetPressureSlave1 := GET_SYNC_REFTO('Pump1.sv_KHW_ServoSlave1_setValue.rAux[1]', T#0s, Status);
   mprSetVelocitySlave1 := GET_SYNC_REFTO('Pump1.sv_KHW_ServoSlave1_setValue.rVeloc', T#0s, Status);
   mpSlave1State := GET_SYNC_REFTO("Pump1.sv_KHW_ServoSlave1_state_sim", T#0s, Status);
   IF Status <> KSYS_Status_OK THEN
      mpSlave1State := GET_SYNC_REFTO("Pump1.sv_KHW_ServoSlave1_state", T#0s, Status);
   END_IF;
   mprActVelocitySlave1 := GET_SYNC_REFTO("Pump1.sv_rActVelocitySlave1", t#0s, Status);
   mpiDriveStatusSlave1 := GET_SYNC_REFTO("Pump1.sv_iDriveStatusSlave1", t#0s, Status);
   mpsRevisionSlave1 := GET_SYNC_REFTO("Pump1.sv_sRevisionSlave1", t#0s, Status);
   mpsDrvIDSlave1 := GET_SYNC_REFTO("Pump1.sv_sDrvID_Slave1", t#0s, Status);
   mprTorqueSlave1 := GET_SYNC_REFTO("Pump1.sv_rMotorTorqueSlave1", T#0s, Status);
   mprMotorPowerSlave1 := GET_SYNC_REFTO("Pump1.sv_rMotorPowerSlave1", T#0s, Status);
END_IF;

(*Slave2*)
IF mbSlave2Linked THEN
   mprSetPressureSlave2 := GET_SYNC_REFTO('Pump1.sv_KHW_ServoSlave2_setValue.rAux[1]', T#0s, Status);
   mprSetVelocitySlave2 := GET_SYNC_REFTO('Pump1.sv_KHW_ServoSlave2_setValue.rVeloc', T#0s, Status);
   mpSlave2State := GET_SYNC_REFTO("Pump1.sv_KHW_ServoSlave2_state_sim", T#0s, Status);
   IF Status <> KSYS_Status_OK THEN
      mpSlave2State := GET_SYNC_REFTO("Pump1.sv_KHW_ServoSlave2_state", T#0s, Status);
   END_IF;
   mprActVelocitySlave2 := GET_SYNC_REFTO("Pump1.sv_rActVelocitySlave2", t#0s, Status);
   mpiDriveStatusSlave2 := GET_SYNC_REFTO("Pump1.sv_iDriveStatusSlave2", t#0s, Status);
   mpsRevisionSlave2 := GET_SYNC_REFTO("Pump1.sv_sRevisionSlave2", t#0s, Status);
   mpsDrvIDSlave2:= GET_SYNC_REFTO("Pump1.sv_sDrvID_Slave2", t#0s, Status);
   mprTorqueSlave2 := GET_SYNC_REFTO("Pump1.sv_rMotorTorqueSlave2", T#0s, Status);
   mprMotorPowerSlave2 := GET_SYNC_REFTO("Pump1.sv_rMotorPowerSlave2", T#0s, Status);
END_IF;

dCycleTime := GET_TASK_INTERVAL();
rCycleTime := (LINT_TO_REAL(TIME_TO_LINT(dCycleTime))) / 1000000.0;

@SaText @RT(9)aStopSimu 1 @TL(7)
(**************************************** WARNING ********************************************
 *** The KEBA Kemro K2 System including software is not intended for safety control tasks! ***
 ***                       For further information see Comment tab!                        ***
 *********************************************************************************************)

STOP_PROCESS_ALGORITHM();

@SaText @RT(9)aSimulate 1 @TL(78)
(**************************************** WARNING ********************************************
 *** The KEBA Kemro K2 System including software is not intended for safety control tasks! ***
 ***                       For further information see Comment tab!                        ***
 *********************************************************************************************)

(*Get the feedback directly from the set values in case of simulation mode*)
(*scaling : 1000% -> 100%*)
rActPressureMaster := mprSetPressureMaster^ / 10.0;
rActVelocityMaster := mprSetVelocityMaster^ / 10.0;
IF mbSlave1Linked THEN
   rActPressureSlave1 := mprSetPressureSlave1^ / 10.0;
   rActVelocitySlave1 := mprSetVelocitySlave1^ / 10.0;
END_IF;
IF mbSlave2Linked THEN
   rActPressureSlave2 := mprSetPressureSlave2^ / 10.0;
   rActVelocitySlave2 := mprSetVelocitySlave2^ / 10.0;
END_IF;

(*Velocity simulation*)
b := WRITE_SVREAL_DIRECT(mprActVelocityMaster^, (rMaxVelocity * rActVelocityMaster  / 100.0 * 30.0 / cApplPlasticsPI)); (*in rpm*)
IF mbSlave1Linked THEN
   b := WRITE_SVREAL_DIRECT(mprActVelocitySlave1^, (rMaxVelocity * rActVelocitySlave1  / 100.0 * 30.0 / cApplPlasticsPI)); (*in rpm*)
END_IF;
IF mbSlave2Linked THEN
   b := WRITE_SVREAL_DIRECT(mprActVelocitySlave2^, (rMaxVelocity * rActVelocitySlave2  / 100.0 * 30.0 / cApplPlasticsPI)); (*in rpm*)
END_IF;

(*Limitation of acceleration in simulation*)
IF rCycleTime <> 0.0 THEN
   mrAccelerationMaster := LIMIT(-14000.0, (rActVelocityMaster - rLastVelocityMaster) /100.0 * rMaxVelocity / rCycleTime, 14000.0);
   IF mbSlave1Linked THEN
      mrAccelerationSlave1 := LIMIT(-14000.0, (rActVelocitySlave1 - rLastVelocitySlave1) /100.0 * rMaxVelocity / rCycleTime, 14000.0);
   END_IF;
   IF mbSlave2Linked THEN
      mrAccelerationSlave2 := LIMIT(-14000.0, (rActVelocitySlave2 - rLastVelocitySlave2) /100.0 * rMaxVelocity / rCycleTime, 14000.0);
   END_IF;
END_IF;

(*100ms as cycle time for torque and power updating*)
IF miCount = 25 THEN
   (* simulate the motor torque *)
   IF mpbInjectionActive^ THEN
      (* pressure-proptional torque is simulated only during injection *)
      b := WRITE_SVREAL_DIRECT(mprTorqueMaster^, (k1 * mrAccelerationMaster + k2 * rActPressureMaster / 100.0 * rMaxPressure + k3 * rActVelocityMaster / 100.0 * rMaxVelocity + rLoadTorque));
      IF mbSlave1Linked THEN
         b := WRITE_SVREAL_DIRECT(mprTorqueSlave1^, (k1 * mrAccelerationSlave1 + k2 * rActPressureSlave1 / 100.0 * rMaxPressure + k3 * rActVelocitySlave1 / 100.0 * rMaxVelocity + rLoadTorque));
      END_IF;
      IF mbSlave2Linked THEN
         b := WRITE_SVREAL_DIRECT(mprTorqueSlave2^, (k1 * mrAccelerationSlave2 + k2 * rActPressureSlave2 / 100.0 * rMaxPressure + k3 * rActVelocitySlave2 / 100.0 * rMaxVelocity + rLoadTorque));
      END_IF;
   ELSE
      b := WRITE_SVREAL_DIRECT(mprTorqueMaster^, (k1 * mrAccelerationMaster + k3 * rActVelocityMaster / 100.0 * rMaxVelocity + rLoadTorque));
      IF mbSlave1Linked THEN
         b := WRITE_SVREAL_DIRECT(mprTorqueSlave1^, (k1 * mrAccelerationSlave1 + k3 * rActVelocitySlave1 / 100.0 * rMaxVelocity + rLoadTorque));
      END_IF;
      IF mbSlave2Linked THEN
         b := WRITE_SVREAL_DIRECT(mprTorqueSlave2^, (k1 * mrAccelerationSlave2 + k3 * rActVelocitySlave2 / 100.0 * rMaxVelocity + rLoadTorque));
      END_IF;
   END_IF;

   (* simulate motor power *)
   b := WRITE_SVREAL_DIRECT(mprMotorPowerMaster^, (mprTorqueMaster^ * rActVelocityMaster / 100.0 * rMaxVelocity / 1000.0));
   IF mbSlave1Linked THEN
      b := WRITE_SVREAL_DIRECT(mprMotorPowerSlave1^, (mprTorqueSlave1^ * rActVelocitySlave1 / 100.0 * rMaxVelocity / 1000.0));
   END_IF;
   IF mbSlave2Linked THEN
      b := WRITE_SVREAL_DIRECT(mprMotorPowerSlave2^, (mprTorqueSlave2^ * rActVelocitySlave2 / 100.0 * rMaxVelocity / 1000.0));
   END_IF;

   miCount := 0;
ELSE
   miCount := miCount + 1;
END_IF;

rLastVelocityMaster := rActVelocityMaster;
rLastVelocitySlave1 := rActVelocitySlave1;
rLastVelocitySlave2 := rActVelocitySlave2;

@SaText @RT(14)aReadDriveInfo 1 @TL(18)
(**************************************** WARNING ********************************************
 *** The KEBA Kemro K2 System including software is not intended for safety control tasks! ***
 ***                       For further information see Comment tab!                        ***
 *********************************************************************************************)

b := WRITE_SV_DIRECT(mpsRevisionMaster^, sRevisionMaster);
b := WRITE_SV_DIRECT(mpsDrvIDMaster^, sDrvIDMaster);

IF mbSlave1Linked THEN
   b := WRITE_SV_DIRECT(mpsRevisionSlave1^, sRevisionMaster);
   b := WRITE_SV_DIRECT(mpsDrvIDSlave1^, sDrvIDMaster);
END_IF;

IF mbSlave2Linked THEN
   b := WRITE_SV_DIRECT(mpsRevisionSlave2^, sRevisionMaster);
   b := WRITE_SV_DIRECT(mpsDrvIDSlave2^, sDrvIDMaster);
END_IF;

@SaTrans 0
@SaExits 0
@END_SfcBody

@@@BEG_Comment@@@
@TL(0)

@@@END_Comment@@@

@BEG_Body
@TL(24)
(**************************************** WARNING ********************************************
 *** The KEBA Kemro K2 System including software is not intended for safety control tasks! ***
 ***                       For further information see Comment tab!                        ***
 *********************************************************************************************)

IF NOT bInitDone THEN
   (*Check if the speed pump exists, simulation will not be started in case of no speedpump*)
   pOptions := GET_SYNC_REFTO('Pump1.sv_Options', T#0s, s);
   mbSpeedPump := (s = KSYS_Status_OK) AND ((pOptions^ AND cSubOpSpeedpumpMaster) = cSubOpSpeedpumpMaster);

   IF ((pOptions^ AND cSubOpSpeedpumpSlave2) = cSubOpSpeedpumpSlave2) THEN
      mbSlave1Linked := TRUE;
      mbSlave2Linked := TRUE;
   ELSIF ((pOptions^ AND cSubOpSpeedpumpSlave1) = cSubOpSpeedpumpSlave1) THEN
      mbSlave1Linked := TRUE;
   END_IF;

   bInitDone := TRUE;
END_IF;

IF sv_bSimulate AND mbSpeedPump THEN
   START_PROCESS_ALGORITHM(paSimulate);
END_IF;

@END_Body

@@@BEG_Comment@@@
@TL(0)

@@@END_Comment@@@

@BEG_Body
@TL(44)
(**************************************** WARNING ********************************************
 *** The KEBA Kemro K2 System including software is not intended for safety control tasks! ***
 ***                       For further information see Comment tab!                        ***
 *********************************************************************************************)
IF mbSpeedPump THEN

   bOnOff := FALSE;

   IF mpbKeyOnOff <> EMPTY THEN
      bOnOff := mpbKeyOnOff^;
   END_IF;

   IF mpbKeyOnOffHMI <> EMPTY THEN
      bOnOff := bOnOff OR mpbKeyOnOffHMI^;
   END_IF;

   IF (bOnOff OR mpbMotorLocked^) THEN
      mbMotorOnReq := (NOT mbMotorOnReq) AND (NOT mpbMotorLocked^);
   END_IF;

   (*Force the status word when motor is shut on or off,
   so that the state handler works in simulation mode*)
   IF mbMotorOnReq THEN
      DriveState := 16#27;
      iDriveStatus := 2;
   ELSE
      DriveState := 0;
      iDriveStatus := 1;
   END_IF;

   mpMasterState^ := DriveState;
   mpiDriveStatusMaster^ := iDriveStatus;

   IF mbSlave1Linked THEN
      mpSlave1State^ := DriveState;
      mpiDriveStatusSlave1^ := iDriveStatus;
   END_IF;

   IF mbSlave2Linked THEN
      mpSlave2State^ := DriveState;
      mpiDriveStatusSlave2^ := iDriveStatus;
   END_IF;
END_IF;

@END_Body

@@@BEG_Comment@@@
@TL(0)

@@@END_Comment@@@

@BEG_Body
@TL(18)
(**************************************** WARNING ********************************************
 *** The KEBA Kemro K2 System including software is not intended for safety control tasks! ***
 ***                       For further information see Comment tab!                        ***
 *********************************************************************************************)

fuName := GET_MY_FU_NAME();
variableName := CONCAT(fuName,'.rTorque Nm');
swoState := KSWO_AddVariable( Task := TaskInject,
                              Name := variableName,
                              Variable := mprTorqueMaster^);

variableName := CONCAT(fuName,'.rAcc rad/s/s');
swoState := KSWO_AddVariable( Task := TaskInject,
                              Name := variableName,
                              Variable := mrAccelerationMaster);
STOP_PROCESS_ALGORITHM();

@END_Body

@@@BEG_Comment@@@
@TL(0)

@@@END_Comment@@@
@END_Body

@END_Contents
